LIN {X 0,Y 193.607,Z 643.258,A -85,B 0,C 180,E1 -26158.912,E2 -26158.912} C_VEL
LIN {X 0,Y 201.714,Z 651.879,A -85,B 0,C 180,E1 -26162.725,E2 -26162.725} C_VEL
LIN {X 0,Y 211.086,Z 659.54,A -85,B 0,C 180,E1 -26166.451,E2 -26166.451} C_VEL
LIN {X 0,Y 220.948,Z 665.783,A -85,B 0,C 180,E1 -26169.763,E2 -26169.763} C_VEL
LIN {X 0,Y 234.366,Z 672.498,A -85,B 0,C 180,E1 -26173.645,E2 -26173.645} C_VEL
LIN {X 0,Y 246.298,Z 677.555,A -85,B 0,C 180,E1 -26176.805,E2 -26176.805} C_VEL
LIN {X 0,Y 253.834,Z 680.558,A -85,B 0,C 180,E1 -26178.825,E2 -26178.825} C_VEL
LIN {X 0,Y 260.206,Z 683.111,A -85,B 0,C 180,E1 -26180.674,E2 -26180.674} C_VEL
LIN {X 0,Y 265.463,Z 685.211,A -85,B 0,C 180,E1 -26182.393,E2 -26182.393} C_VEL
LIN {X 0,Y 269.417,Z 686.886,A -85,B 0,C 180,E1 -26184.011,E2 -26184.011} C_VEL
LIN {X 0,Y 272.304,Z 688.198,A -85,B 0,C 180,E1 -26185.559,E2 -26185.559} C_VEL
LIN {X 0,Y 274.956,Z 689.105,A -85,B 0,C 180,E1 -26187.07,E2 -26187.07} C_VEL
LIN {X 0,Y 276.564,Z 689.664,A -85,B 0,C 180,E1 -26188.544,E2 -26188.544} C_VEL
LIN {X 0,Y 277.483,Z 689.842,A -85,B 0,C 180,E1 -26190,E2 -26190} C_VEL
LIN {X 0,Y 276.566,Z 689.663,A -85,B 0,C 180,E1 -26191.456,E2 -26191.456} C_VEL
LIN {X 0,Y 274.501,Z 688.974,A -85,B 0,C 180,E1 -26193.184,E2 -26193.184} C_VEL
LIN {X 0,Y 272.278,Z 688.199,A -85,B 0,C 180,E1 -26194.441,E2 -26194.441} C_VEL
LIN {X 0,Y 268.678,Z 686.595,A -85,B 0,C 180,E1 -26196.311,E2 -26196.311} C_VEL
LIN {X 0,Y 265.415,Z 685.213,A -85,B 0,C 180,E1 -26197.608,E2 -26197.608} C_VEL
LIN {X 0,Y 260.173,Z 683.112,A -85,B 0,C 180,E1 -26199.327,E2 -26199.327} C_VEL
LIN {X 0,Y 253.886,Z 680.557,A -85,B 0,C 180,E1 -26201.173,E2 -26201.173} C_VEL
LIN {X 0,Y 245.609,Z 677.259,A -85,B 0,C 180,E1 -26203.385,E2 -26203.385} C_VEL
LIN {X 0,Y 234.359,Z 672.513,A -85,B 0,C 180,E1 -26206.349,E2 -26206.349} C_VEL
LIN {X 0,Y 220.948,Z 665.784,A -85,B 0,C 180,E1 -26210.237,E2 -26210.237} C_VEL
LIN {X 0,Y 211.166,Z 659.537,A -85,B 0,C 180,E1 -26213.539,E2 -26213.539} C_VEL
LIN {X 0,Y 201.751,Z 651.903,A -85,B 0,C 180,E1 -26217.262,E2 -26217.262} C_VEL
LIN {X 0,Y 192.245,Z 641.559,A -85,B 0,C 180,E1 -26221.794,E2 -26221.794} C_VEL
LIN {X 0,Y 185.61,Z 632.244,A -85,B 0,C 180,E1 -26225.461,E2 -26225.461} C_VEL
LIN {X 0,Y 180.259,Z 622.941,A -85,B 0,C 180,E1 -26228.767,E2 -26228.767} C_VEL
LIN {X 0,Y 175.258,Z 612.247,A -85,B 0,C 180,E1 -26232.116,E2 -26232.116} C_VEL
LIN {X 0,Y 170.985,Z 601.587,A -85,B 0,C 180,E1 -26235.058,E2 -26235.058} C_VEL
LIN {X 0,Y 167.177,Z 590.937,A -85,B 0,C 180,E1 -26237.634,E2 -26237.634} C_VEL
LIN {X 0,Y 160.92,Z 572.907,A -85,B 0,C 180,E1 -26241.531,E2 -26241.531} C_VEL
LIN {X 0,Y 157.524,Z 564.607,A -85,B 0,C 180,E1 -26243.75,E2 -26243.75} C_VEL
LIN {X 0,Y 153.292,Z 555.729,A -85,B 0,C 180,E1 -26246.722,E2 -26246.722} C_VEL
LIN {X 0,Y 148.61,Z 547.106,A -85,B 0,C 180,E1 -26250.427,E2 -26250.427} C_VEL
LIN {X 0,Y 144.239,Z 539.962,A -85,B 0,C 180,E1 -26254.48,E2 -26254.48} C_VEL
LIN {X 0,Y 141.462,Z 535.851,A -85,B 0,C 180,E1 -26257.504,E2 -26257.504} C_VEL
LIN {X 0,Y 138.867,Z 531.989,A -85,B 0,C 180,E1 -26260.874,E2 -26260.874} C_VEL
LIN {X 0,Y 136.38,Z 528.521,A -85,B 0,C 180,E1 -26264.882,E2 -26264.882} C_VEL
LIN {X 0,Y 135.759,Z 527.362,A -85,B 0,C 180,E1 -26266.152,E2 -26266.152} C_VEL
LIN {X 0,Y 133.331,Z 524.419,A -85,B 0,C 180,E1 -26272.623,E2 -26272.623} C_VEL
LIN {X 0,Y 132.769,Z 522.602,A -85,B 0,C 180,E1 -26276.211,E2 -26276.211} C_VEL
LIN {X 0,Y 132.584,Z 521.985,A -85,B 0,C 180,E1 -26280.005,E2 -26280.005} C_VEL
LIN {X 0,Y 132.854,Z 522.928,A -85,B 0,C 180,E1 -26284.176,E2 -26284.176} C_VEL
LIN {X 0,Y 135.306,Z 527.03,A -85,B 0,C 180,E1 -26292.567,E2 -26292.567} C_VEL
LIN {X 0,Y 136.125,Z 527.942,A -85,B 0,C 180,E1 -26294.2,E2 -26294.2} C_VEL
LIN {X 0,Y 138.548,Z 531.658,A -85,B 0,C 180,E1 -26298.297,E2 -26298.297} C_VEL
LIN {X 0,Y 139.546,Z 533.014,A -85,B 0,C 180,E1 -26299.687,E2 -26299.687} C_VEL
LIN {X 0,Y 142.466,Z 537.271,A -85,B 0,C 180,E1 -26303.248,E2 -26303.248} C_VEL
LIN {X 0,Y 145.553,Z 542.106,A -85,B 0,C 180,E1 -26306.436,E2 -26306.436} C_VEL
LIN {X 0,Y 147.873,Z 546.115,A -85,B 0,C 180,E1 -26308.575,E2 -26308.575} C_VEL
LIN {X 0,Y 151.392,Z 554.209,A -85,B 0,C 180,E1 -26311.634,E2 -26311.634} C_VEL
LIN {X 0,Y 155.275,Z 564.625,A -85,B 0,C 180,E1 -26314.706,E2 -26314.706} C_VEL
LIN {X 0,Y 156.576,Z 568.776,A -85,B 0,C 180,E1 -26315.702,E2 -26315.702} C_VEL
LIN {X 0,Y 154.246,Z 595.965,A -85,B 0,C 180,E1 -26316.746,E2 -26316.746} C_VEL
LIN {X 0,Y 152.545,Z 606.818,A -85,B 0,C 180,E1 -26317.392,E2 -26317.392} C_VEL
LIN {X 0,Y 150.313,Z 616.609,A -85,B 0,C 180,E1 -26318.18,E2 -26318.18} C_VEL
LIN {X 0,Y 147.465,Z 626.405,A -85,B 0,C 180,E1 -26319.245,E2 -26319.245} C_VEL
LIN {X 0,Y 144.346,Z 635.167,A -85,B 0,C 180,E1 -26320.47,E2 -26320.47} C_VEL
LIN {X 0,Y 140.701,Z 643.886,A -85,B 0,C 180,E1 -26322.013,E2 -26322.013} C_VEL
LIN {X 0,Y 136.637,Z 652.394,A -85,B 0,C 180,E1 -26323.938,E2 -26323.938} C_VEL
LIN {X 0,Y 132.209,Z 660.562,A -85,B 0,C 180,E1 -26326.287,E2 -26326.287} C_VEL
LIN {X 0,Y 128.06,Z 667.504,A -85,B 0,C 180,E1 -26328.81,E2 -26328.81} C_VEL
LIN {X 0,Y 124.167,Z 673.491,A -85,B 0,C 180,E1 -26331.493,E2 -26331.493} C_VEL
LIN {X 0,Y 119.546,Z 680.2,A -85,B 0,C 180,E1 -26335.399,E2 -26335.399} C_VEL
LIN {X 0,Y 116.001,Z 685.08,A -85,B 0,C 180,E1 -26339.004,E2 -26339.004} C_VEL
LIN {X 0,Y 111.98,Z 690.174,A -85,B 0,C 180,E1 -26343.939,E2 -26343.939} C_VEL
LIN {X 0,Y 108.812,Z 694.141,A -85,B 0,C 180,E1 -26349.192,E2 -26349.192} C_VEL
LIN {X 0,Y 106.71,Z 697.085,A -85,B 0,C 180,E1 -26354.726,E2 -26354.726} C_VEL
LIN {X 0,Y 105.784,Z 698.592,A -85,B 0,C 180,E1 -26358.503,E2 -26358.503} C_VEL
LIN {X 0,Y 105.043,Z 700.131,A -85,B 0,C 180,E1 -26366.164,E2 -26366.164} C_VEL
LIN {X 0,Y 105.176,Z 700.418,A -85,B 0,C 180,E1 -26370,E2 -26370} C_VEL
LIN {X 0,Y 105.231,Z 699.528,A -85,B 0,C 180,E1 -26377.676,E2 -26377.676} C_VEL
LIN {X 0,Y 105.787,Z 698.592,A -85,B 0,C 180,E1 -26381.496,E2 -26381.496} C_VEL
LIN {X 0,Y 107.993,Z 695.232,A -85,B 0,C 180,E1 -26388.989,E2 -26388.989} C_VEL
LIN {X 0,Y 110.82,Z 691.602,A -85,B 0,C 180,E1 -26394.344,E2 -26394.344} C_VEL
LIN {X 0,Y 114.515,Z 686.868,A -85,B 0,C 180,E1 -26399.404,E2 -26399.404} C_VEL
LIN {X 0,Y 118.575,Z 681.494,A -85,B 0,C 180,E1 -26403.708,E2 -26403.708} C_VEL
LIN {X 0,Y 122.392,Z 676.116,A -85,B 0,C 180,E1 -26407.08,E2 -26407.08} C_VEL
LIN {X 0,Y 126.08,Z 670.624,A -85,B 0,C 180,E1 -26409.869,E2 -26409.869} C_VEL
LIN {X 0,Y 131.15,Z 662.411,A -85,B 0,C 180,E1 -26413.097,E2 -26413.097} C_VEL
LIN {X 0,Y 135.553,Z 654.591,A -85,B 0,C 180,E1 -26415.47,E2 -26415.47} C_VEL
LIN {X 0,Y 139.541,Z 646.511,A -85,B 0,C 180,E1 -26417.441,E2 -26417.441} C_VEL
LIN {X 0,Y 143.721,Z 636.756,A -85,B 0,C 180,E1 -26419.284,E2 -26419.284} C_VEL
LIN {X 0,Y 146.789,Z 628.37,A -85,B 0,C 180,E1 -26420.536,E2 -26420.536} C_VEL
LIN {X 0,Y 149.971,Z 617.87,A -85,B 0,C 180,E1 -26421.715,E2 -26421.715} C_VEL
LIN {X 0,Y 152.398,Z 607.507,A -85,B 0,C 180,E1 -26422.571,E2 -26422.571} C_VEL
LIN {X 0,Y 154.029,Z 597.554,A -85,B 0,C 180,E1 -26423.182,E2 -26423.182} C_VEL
LIN {X 0,Y 155.824,Z 578.344,A -85,B 0,C 180,E1 -26423.944,E2 -26423.944} C_VEL
LIN {X 0,Y 156.52,Z 568.606,A -85,B 0,C 180,E1 -26424.339,E2 -26424.339} C_VEL
LIN {X 0,Y 153.874,Z 560.714,A -85,B 0,C 180,E1 -26426.368,E2 -26426.368} C_VEL
LIN {X 0,Y 149.72,Z 550.16,A -85,B 0,C 180,E1 -26429.786,E2 -26429.786} C_VEL
LIN {X 0,Y 147.011,Z 544.436,A -85,B 0,C 180,E1 -26432.214,E2 -26432.214} C_VEL
LIN {X 0,Y 143.831,Z 539.389,A -85,B 0,C 180,E1 -26435.281,E2 -26435.281} C_VEL
LIN {X 0,Y 141.559,Z 535.941,A -85,B 0,C 180,E1 -26437.786,E2 -26437.786} C_VEL
LIN {X 0,Y 139.135,Z 532.246,A -85,B 0,C 180,E1 -26440.903,E2 -26440.903} C_VEL
LIN {X 0,Y 138.064,Z 531.159,A -85,B 0,C 180,E1 -26442.398,E2 -26442.398} C_VEL
LIN {X 0,Y 136.969,Z 530.727,A -85,B 0,C 180,E1 -26443.964,E2 -26443.964} C_VEL
LIN {X 0,Y 134.922,Z 531.049,A -85,B 0,C 180,E1 -26447.206,E2 -26447.206} C_VEL
LIN {X 0,Y 133.264,Z 531.693,A -85,B 0,C 180,E1 -26450.577,E2 -26450.577} C_VEL
LIN {X 0,Y 132.425,Z 531.436,A -85,B 0,C 180,E1 -26453.142,E2 -26453.142} C_VEL
LIN {X 0,Y 132.241,Z 531.075,A -85,B 0,C 180,E1 -26453.991,E2 -26453.991} C_VEL
LIN {X 0,Y 131.799,Z 529.387,A -85,B 0,C 180,E1 -26457.703,E2 -26457.703} C_VEL
LIN {X 0,Y 131.717,Z 529.047,A -85,B 0,C 180,E1 -26459.995,E2 -26459.995} C_VEL
LIN {X 0,Y 131.926,Z 529.956,A -85,B 0,C 180,E1 -26464.196,E2 -26464.196} C_VEL
LIN {X 0,Y 134.158,Z 533.971,A -85,B 0,C 180,E1 -26472.428,E2 -26472.428} C_VEL
LIN {X 0,Y 134.782,Z 534.696,A -85,B 0,C 180,E1 -26473.758,E2 -26473.758} C_VEL
LIN {X 0,Y 137.254,Z 538.568,A -85,B 0,C 180,E1 -26478.18,E2 -26478.18} C_VEL
LIN {X 0,Y 140.569,Z 543.731,A -85,B 0,C 180,E1 -26482.647,E2 -26482.647} C_VEL
LIN {X 0,Y 143.405,Z 548.348,A -85,B 0,C 180,E1 -26485.777,E2 -26485.777} C_VEL
LIN {X 0,Y 147.758,Z 556.106,A -85,B 0,C 180,E1 -26489.858,E2 -26489.858} C_VEL
LIN {X 0,Y 152.402,Z 565.552,A -85,B 0,C 180,E1 -26493.594,E2 -26493.594} C_VEL
LIN {X 0,Y 156.256,Z 574.926,A -85,B 0,C 180,E1 -26496.401,E2 -26496.401} C_VEL
LIN {X 0,Y 160.04,Z 586.179,A -85,B 0,C 180,E1 -26499.036,E2 -26499.036} C_VEL
LIN {X 0,Y 163.433,Z 597.185,A -85,B 0,C 180,E1 -26501.588,E2 -26501.588} C_VEL
LIN {X 0,Y 166.658,Z 607.047,A -85,B 0,C 180,E1 -26504.202,E2 -26504.202} C_VEL
LIN {X 0,Y 170.411,Z 617.155,A -85,B 0,C 180,E1 -26507.266,E2 -26507.266} C_VEL
LIN {X 0,Y 174.824,Z 627.17,A -85,B 0,C 180,E1 -26510.695,E2 -26510.695} C_VEL
LIN {X 0,Y 179.681,Z 635.973,A -85,B 0,C 180,E1 -26514.077,E2 -26514.077} C_VEL
LIN {X 0,Y 184.854,Z 643.572,A -85,B 0,C 180,E1 -26517.273,E2 -26517.273} C_VEL
LIN {X 0,Y 192.277,Z 652.277,A -85,B 0,C 180,E1 -26521.302,E2 -26521.302} C_VEL
LIN {X 0,Y 200.736,Z 659.845,A -85,B 0,C 180,E1 -26525.157,E2 -26525.157} C_VEL
LIN {X 0,Y 210.803,Z 666.663,A -85,B 0,C 180,E1 -26528.976,E2 -26528.976} C_VEL
LIN {X 0,Y 221.28,Z 672.126,A -85,B 0,C 180,E1 -26532.318,E2 -26532.318} C_VEL
LIN {X 0,Y 235.082,Z 677.867,A -85,B 0,C 180,E1 -26536.163,E2 -26536.163} C_VEL
LIN {X 0,Y 246.752,Z 682.108,A -85,B 0,C 180,E1 -26539.288,E2 -26539.288} C_VEL
LIN {X 0,Y 255.57,Z 685.165,A -85,B 0,C 180,E1 -26541.858,E2 -26541.858} C_VEL
LIN {X 0,Y 261.463,Z 687.257,A -85,B 0,C 180,E1 -26543.981,E2 -26543.981} C_VEL
LIN {X 0,Y 264.432,Z 688.418,A -85,B 0,C 180,E1 -26545.427,E2 -26545.427} C_VEL
LIN {X 0,Y 267.399,Z 689.359,A -85,B 0,C 180,E1 -26547.069,E2 -26547.069} C_VEL
LIN {X 0,Y 269.242,Z 689.867,A -85,B 0,C 180,E1 -26548.504,E2 -26548.504} C_VEL
LIN {X 0,Y 270.315,Z 690.041,A -85,B 0,C 180,E1 -26550,E2 -26550} C_VEL
LIN {X 0,Y 269.24,Z 689.867,A -85,B 0,C 180,E1 -26551.496,E2 -26551.496} C_VEL
LIN {X 0,Y 267.239,Z 689.317,A -85,B 0,C 180,E1 -26553.015,E2 -26553.015} C_VEL
LIN {X 0,Y 264.41,Z 688.418,A -85,B 0,C 180,E1 -26554.574,E2 -26554.574} C_VEL
LIN {X 0,Y 261.016,Z 687.117,A -85,B 0,C 180,E1 -26556.183,E2 -26556.183} C_VEL
LIN {X 0,Y 255.564,Z 685.178,A -85,B 0,C 180,E1 -26558.132,E2 -26558.132} C_VEL
LIN {X 0,Y 249.679,Z 683.135,A -85,B 0,C 180,E1 -26559.893,E2 -26559.893} C_VEL
LIN {X 0,Y 243.252,Z 680.857,A -85,B 0,C 180,E1 -26561.668,E2 -26561.668} C_VEL
LIN {X 0,Y 232.346,Z 676.846,A -85,B 0,C 180,E1 -26564.562,E2 -26564.562} C_VEL
LIN {X 0,Y 217.434,Z 670.286,A -85,B 0,C 180,E1 -26568.858,E2 -26568.858} C_VEL
LIN {X 0,Y 205.884,Z 663.53,A -85,B 0,C 180,E1 -26572.839,E2 -26572.839} C_VEL
LIN {X 0,Y 195.479,Z 655.394,A -85,B 0,C 180,E1 -26577.158,E2 -26577.158} C_VEL
LIN {X 0,Y 188.212,Z 647.778,A -85,B 0,C 180,E1 -26580.821,E2 -26580.821} C_VEL
LIN {X 0,Y 181.58,Z 639.028,A -85,B 0,C 180,E1 -26584.674,E2 -26584.674} C_VEL
LIN {X 0,Y 176.615,Z 630.661,A -85,B 0,C 180,E1 -26588.007,E2 -26588.007} C_VEL
LIN {X 0,Y 172.513,Z 622.049,A -85,B 0,C 180,E1 -26591.095,E2 -26591.095} C_VEL
LIN {X 0,Y 168.754,Z 612.855,A -85,B 0,C 180,E1 -26594.083,E2 -26594.083} C_VEL
LIN {X 0,Y 164.892,Z 601.852,A -85,B 0,C 180,E1 -26597.218,E2 -26597.218} C_VEL
LIN {X 0,Y 161.241,Z 590.184,A -85,B 0,C 180,E1 -26600.098,E2 -26600.098} C_VEL
LIN {X 0,Y 156.857,Z 576.56,A -85,B 0,C 180,E1 -26603.178,E2 -26603.178} C_VEL
LIN {X 0,Y 152.863,Z 566.622,A -85,B 0,C 180,E1 -26606.056,E2 -26606.056} C_VEL
LIN {X 0,Y 148.504,Z 557.612,A -85,B 0,C 180,E1 -26609.499,E2 -26609.499} C_VEL
LIN {X 0,Y 144.243,Z 549.708,A -85,B 0,C 180,E1 -26613.387,E2 -26613.387} C_VEL
LIN {X 0,Y 141.473,Z 545.217,A -85,B 0,C 180,E1 -26616.297,E2 -26616.297} C_VEL
LIN {X 0,Y 139.46,Z 542.029,A -85,B 0,C 180,E1 -26618.719,E2 -26618.719} C_VEL
LIN {X 0,Y 137.255,Z 538.56,A -85,B 0,C 180,E1 -26621.819,E2 -26621.819} C_VEL
LIN {X 0,Y 134.781,Z 534.7,A -85,B 0,C 180,E1 -26626.242,E2 -26626.242} C_VEL
LIN {X 0,Y 134.159,Z 533.961,A -85,B 0,C 180,E1 -26627.572,E2 -26627.572} C_VEL
LIN {X 0,Y 131.822,Z 529.519,A -85,B 0,C 180,E1 -26636.949,E2 -26636.949} C_VEL
LIN {X 0,Y 131.718,Z 529.04,A -85,B 0,C 180,E1 -26640.005,E2 -26640.005} C_VEL
LIN {X 0,Y 131.94,Z 529.991,A -85,B 0,C 180,E1 -26643.918,E2 -26643.918} C_VEL
LIN {X 0,Y 134.319,Z 534.061,A -85,B 0,C 180,E1 -26652.373,E2 -26652.373} C_VEL
LIN {X 0,Y 134.87,Z 534.887,A -85,B 0,C 180,E1 -26653.566,E2 -26653.566} C_VEL
LIN {X 0,Y 137.881,Z 539.509,A -85,B 0,C 180,E1 -26658.726,E2 -26658.726} C_VEL
LIN {X 0,Y 140.659,Z 543.824,A -85,B 0,C 180,E1 -26662.359,E2 -26662.359} C_VEL
LIN {X 0,Y 144.231,Z 549.666,A -85,B 0,C 180,E1 -26666.21,E2 -26666.21} C_VEL
LIN {X 0,Y 146.772,Z 555.356,A -85,B 0,C 180,E1 -26668.712,E2 -26668.712} C_VEL
LIN {X 0,Y 150.791,Z 566.153,A -85,B 0,C 180,E1 -26672.316,E2 -26672.316} C_VEL
LIN {X 0,Y 152.326,Z 571.077,A -85,B 0,C 180,E1 -26673.622,E2 -26673.622} C_VEL
LIN {X 0,Y 150.054,Z 596.194,A -85,B 0,C 180,E1 -26674.595,E2 -26674.595} C_VEL
LIN {X 0,Y 148.212,Z 607.312,A -85,B 0,C 180,E1 -26675.26,E2 -26675.26} C_VEL
LIN {X 0,Y 145.05,Z 620.182,A -85,B 0,C 180,E1 -26676.341,E2 -26676.341} C_VEL
LIN {X 0,Y 141.148,Z 631.794,A -85,B 0,C 180,E1 -26677.774,E2 -26677.774} C_VEL
LIN {X 0,Y 136.685,Z 642.378,A -85,B 0,C 180,E1 -26679.533,E2 -26679.533} C_VEL
LIN {X 0,Y 132.432,Z 651.101,A -85,B 0,C 180,E1 -26681.445,E2 -26681.445} C_VEL
LIN {X 0,Y 128.306,Z 658.516,A -85,B 0,C 180,E1 -26683.467,E2 -26683.467} C_VEL
LIN {X 0,Y 122.8,Z 667.308,A -85,B 0,C 180,E1 -26686.625,E2 -26686.625} C_VEL
LIN {X 0,Y 118.669,Z 673.294,A -85,B 0,C 180,E1 -26689.349,E2 -26689.349} C_VEL
LIN {X 0,Y 114.137,Z 679.517,A -85,B 0,C 180,E1 -26693.014,E2 -26693.014} C_VEL
LIN {X 0,Y 109.963,Z 684.884,A -85,B 0,C 180,E1 -26697.095,E2 -26697.095} C_VEL
LIN {X 0,Y 105.619,Z 689.977,A -85,B 0,C 180,E1 -26702.239,E2 -26702.239} C_VEL
LIN {X 0,Y 102.189,Z 693.944,A -85,B 0,C 180,E1 -26707.774,E2 -26707.774} C_VEL
LIN {X 0,Y 99.835,Z 696.887,A -85,B 0,C 180,E1 -26713.645,E2 -26713.645} C_VEL
LIN {X 0,Y 98.804,Z 698.395,A -85,B 0,C 180,E1 -26717.679,E2 -26717.679} C_VEL
LIN {X 0,Y 97.949,Z 699.935,A -85,B 0,C 180,E1 -26725.885,E2 -26725.885} C_VEL
LIN {X 0,Y 98.083,Z 700.222,A -85,B 0,C 180,E1 -26730,E2 -26730} C_VEL
LIN {X 0,Y 98.188,Z 699.331,A -85,B 0,C 180,E1 -26738.23,E2 -26738.23} C_VEL
LIN {X 0,Y 98.806,Z 698.395,A -85,B 0,C 180,E1 -26742.321,E2 -26742.321} C_VEL
LIN {X 0,Y 101.264,Z 695.034,A -85,B 0,C 180,E1 -26750.305,E2 -26750.305} C_VEL
LIN {X 0,Y 104.361,Z 691.405,A -85,B 0,C 180,E1 -26755.959,E2 -26755.959} C_VEL
LIN {X 0,Y 108.374,Z 686.672,A -85,B 0,C 180,E1 -26761.251,E2 -26761.251} C_VEL
LIN {X 0,Y 113.448,Z 680.404,A -85,B 0,C 180,E1 -26766.349,E2 -26766.349} C_VEL
LIN {X 0,Y 118.685,Z 673.295,A -85,B 0,C 180,E1 -26770.645,E2 -26770.645} C_VEL
LIN {X 0,Y 124.945,Z 664.064,A -85,B 0,C 180,E1 -26774.676,E2 -26774.676} C_VEL
LIN {X 0,Y 130.657,Z 654.394,A -85,B 0,C 180,E1 -26777.697,E2 -26777.697} C_VEL
LIN {X 0,Y 134.838,Z 646.315,A -85,B 0,C 180,E1 -26779.665,E2 -26779.665} C_VEL
LIN {X 0,Y 139.196,Z 636.56,A -85,B 0,C 180,E1 -26781.498,E2 -26781.498} C_VEL
LIN {X 0,Y 142.374,Z 628.173,A -85,B 0,C 180,E1 -26782.747,E2 -26782.747} C_VEL
LIN {X 0,Y 145.686,Z 617.674,A -85,B 0,C 180,E1 -26783.903,E2 -26783.903} C_VEL
LIN {X 0,Y 148.191,Z 607.313,A -85,B 0,C 180,E1 -26784.751,E2 -26784.751} C_VEL
LIN {X 0,Y 149.949,Z 596.931,A -85,B 0,C 180,E1 -26785.365,E2 -26785.365} C_VEL
LIN {X 0,Y 151.985,Z 575.616,A -85,B 0,C 180,E1 -26786.192,E2 -26786.192} C_VEL
LIN {X 0,Y 152.233,Z 570.793,A -85,B 0,C 180,E1 -26786.453,E2 -26786.453} C_VEL
LIN {X 0,Y 150.06,Z 564.182,A -85,B 0,C 180,E1 -26788.299,E2 -26788.299} C_VEL
LIN {X 0,Y 146.442,Z 554.498,A -85,B 0,C 180,E1 -26791.609,E2 -26791.609} C_VEL
LIN {X 0,Y 144.15,Z 549.512,A -85,B 0,C 180,E1 -26793.872,E2 -26793.872} C_VEL
LIN {X 0,Y 140.041,Z 542.737,A -85,B 0,C 180,E1 -26798.404,E2 -26798.404} C_VEL
LIN {X 0,Y 137.085,Z 538.343,A -85,B 0,C 180,E1 -26802.466,E2 -26802.466} C_VEL
LIN {X 0,Y 134.697,Z 534.461,A -85,B 0,C 180,E1 -26806.834,E2 -26806.834} C_VEL
LIN {X 0,Y 132.241,Z 531.075,A -85,B 0,C 180,E1 -26813.991,E2 -26813.991} C_VEL
LIN {X 0,Y 131.928,Z 530.66,A -85,B 0,C 180,E1 -26815.676,E2 -26815.676} C_VEL
LIN {X 0,Y 131.504,Z 531.404,A -85,B 0,C 180,E1 -26818.225,E2 -26818.225} C_VEL
LIN {X 0,Y 131.115,Z 534.724,A -85,B 0,C 180,E1 -26822.391,E2 -26822.391} C_VEL
LIN {X 0,Y 131.269,Z 537.711,A -85,B 0,C 180,E1 -26825.753,E2 -26825.753} C_VEL
LIN {X 0,Y 131.577,Z 538.823,A -85,B 0,C 180,E1 -26827.477,E2 -26827.477} C_VEL
LIN {X 0,Y 133.476,Z 541.439,A -85,B 0,C 180,E1 -26832.926,E2 -26832.926} C_VEL
LIN {X 0,Y 135.862,Z 545.334,A -85,B 0,C 180,E1 -26837.493,E2 -26837.493} C_VEL
LIN {X 0,Y 138.864,Z 550.396,A -85,B 0,C 180,E1 -26841.815,E2 -26841.815} C_VEL
LIN {X 0,Y 141.09,Z 554.185,A -85,B 0,C 180,E1 -26844.455,E2 -26844.455} C_VEL
LIN {X 0,Y 145.036,Z 561.671,A -85,B 0,C 180,E1 -26848.487,E2 -26848.487} C_VEL
LIN {X 0,Y 149.247,Z 570.719,A -85,B 0,C 180,E1 -26852.172,E2 -26852.172} C_VEL
LIN {X 0,Y 152.826,Z 579.943,A -85,B 0,C 180,E1 -26855.011,E2 -26855.011} C_VEL
LIN {X 0,Y 155.977,Z 590.349,A -85,B 0,C 180,E1 -26857.561,E2 -26857.561} C_VEL
LIN {X 0,Y 158.362,Z 599.183,A -85,B 0,C 180,E1 -26859.737,E2 -26859.737} C_VEL
LIN {X 0,Y 161.065,Z 608.7,A -85,B 0,C 180,E1 -26862.383,E2 -26862.383} C_VEL
LIN {X 0,Y 163.883,Z 617.554,A -85,B 0,C 180,E1 -26865.153,E2 -26865.153} C_VEL
LIN {X 0,Y 167.126,Z 626.218,A -85,B 0,C 180,E1 -26868.185,E2 -26868.185} C_VEL
LIN {X 0,Y 170.873,Z 634.482,A -85,B 0,C 180,E1 -26871.389,E2 -26871.389} C_VEL
LIN {X 0,Y 176.446,Z 644.006,A -85,B 0,C 180,E1 -26875.553,E2 -26875.553} C_VEL
LIN {X 0,Y 183.092,Z 652.655,A -85,B 0,C 180,E1 -26879.749,E2 -26879.749} C_VEL
LIN {X 0,Y 190.671,Z 660.146,A -85,B 0,C 180,E1 -26883.749,E2 -26883.749} C_VEL
LIN {X 0,Y 198.336,Z 665.908,A -85,B 0,C 180,E1 -26887.108,E2 -26887.108} C_VEL
LIN {X 0,Y 208.351,Z 671.711,A -85,B 0,C 180,E1 -26890.808,E2 -26890.808} C_VEL
LIN {X 0,Y 219.133,Z 676.52,A -85,B 0,C 180,E1 -26894.173,E2 -26894.173} C_VEL
LIN {X 0,Y 232.109,Z 681.172,A -85,B 0,C 180,E1 -26897.763,E2 -26897.763} C_VEL
LIN {X 0,Y 242.25,Z 684.363,A -85,B 0,C 180,E1 -26900.515,E2 -26900.515} C_VEL
LIN {X 0,Y 248.219,Z 686.173,A -85,B 0,C 180,E1 -26902.274,E2 -26902.274} C_VEL
LIN {X 0,Y 254.236,Z 687.958,A -85,B 0,C 180,E1 -26904.334,E2 -26904.334} C_VEL
LIN {X 0,Y 256.368,Z 688.643,A -85,B 0,C 180,E1 -26905.283,E2 -26905.283} C_VEL
LIN {X 0,Y 260.299,Z 689.748,A -85,B 0,C 180,E1 -26907.356,E2 -26907.356} C_VEL
LIN {X 0,Y 261.821,Z 690.072,A -85,B 0,C 180,E1 -26908.462,E2 -26908.462} C_VEL
LIN {X 0,Y 263.123,Z 690.239,A -85,B 0,C 180,E1 -26910,E2 -26910} C_VEL
LIN {X 0,Y 261.817,Z 690.071,A -85,B 0,C 180,E1 -26911.538,E2 -26911.538} C_VEL
LIN {X 0,Y 259.449,Z 689.531,A -85,B 0,C 180,E1 -26913.106,E2 -26913.106} C_VEL
LIN {X 0,Y 256.345,Z 688.643,A -85,B 0,C 180,E1 -26914.718,E2 -26914.718} C_VEL
LIN {X 0,Y 254.232,Z 687.965,A -85,B 0,C 180,E1 -26915.658,E2 -26915.658} C_VEL
LIN {X 0,Y 248.218,Z 686.176,A -85,B 0,C 180,E1 -26917.724,E2 -26917.724} C_VEL
LIN {X 0,Y 239.977,Z 683.679,A -85,B 0,C 180,E1 -26920.12,E2 -26920.12} C_VEL
LIN {X 0,Y 230.5,Z 680.631,A -85,B 0,C 180,E1 -26922.676,E2 -26922.676} C_VEL
LIN {X 0,Y 214.81,Z 674.704,A -85,B 0,C 180,E1 -26927.125,E2 -26927.125} C_VEL
LIN {X 0,Y 203.242,Z 668.921,A -85,B 0,C 180,E1 -26931,E2 -26931} C_VEL
LIN {X 0,Y 193.666,Z 662.535,A -85,B 0,C 180,E1 -26934.884,E2 -26934.884} C_VEL
LIN {X 0,Y 186.106,Z 655.804,A -85,B 0,C 180,E1 -26938.606,E2 -26938.606} C_VEL
LIN {X 0,Y 179.276,Z 647.971,A -85,B 0,C 180,E1 -26942.568,E2 -26942.568} C_VEL
LIN {X 0,Y 174.048,Z 640.217,A -85,B 0,C 180,E1 -26946.146,E2 -26946.146} C_VEL
LIN {X 0,Y 169.699,Z 632.112,A -85,B 0,C 180,E1 -26949.557,E2 -26949.557} C_VEL
LIN {X 0,Y 165.816,Z 622.857,A -85,B 0,C 180,E1 -26953.025,E2 -26953.025} C_VEL
LIN {X 0,Y 162.519,Z 613.253,A -85,B 0,C 180,E1 -26956.225,E2 -26956.225} C_VEL
LIN {X 0,Y 159.259,Z 602.507,A -85,B 0,C 180,E1 -26959.396,E2 -26959.396} C_VEL
LIN {X 0,Y 156.191,Z 591.08,A -85,B 0,C 180,E1 -26962.296,E2 -26962.296} C_VEL
LIN {X 0,Y 152.909,Z 580.112,A -85,B 0,C 180,E1 -26964.93,E2 -26964.93} C_VEL
LIN {X 0,Y 149.16,Z 570.549,A -85,B 0,C 180,E1 -26967.896,E2 -26967.896} C_VEL
LIN {X 0,Y 145.19,Z 562.04,A -85,B 0,C 180,E1 -26971.363,E2 -26971.363} C_VEL
LIN {X 0,Y 141.548,Z 554.977,A -85,B 0,C 180,E1 -26975.042,E2 -26975.042} C_VEL
LIN {X 0,Y 138.144,Z 549.065,A -85,B 0,C 180,E1 -26979.143,E2 -26979.143} C_VEL
LIN {X 0,Y 135.497,Z 544.882,A -85,B 0,C 180,E1 -26983.09,E2 -26983.09} C_VEL
LIN {X 0,Y 133.157,Z 540.966,A -85,B 0,C 180,E1 -26987.817,E2 -26987.817} C_VEL
LIN {X 0,Y 131.111,Z 537.419,A -85,B 0,C 180,E1 -26995.2,E2 -26995.2} C_VEL
LIN {X 0,Y 130.897,Z 536.44,A -85,B 0,C 180,E1 -26997.697,E2 -26997.697} C_VEL
LIN {X 0,Y 130.857,Z 536.195,A -85,B 0,C 180,E1 -27000.774,E2 -27000.774} C_VEL
LIN {X 0,Y 131.03,Z 537.046,A -85,B 0,C 180,E1 -27003.657,E2 -27003.657} C_VEL
LIN {X 0,Y 133.164,Z 540.952,A -85,B 0,C 180,E1 -27011.805,E2 -27011.805} C_VEL
LIN {X 0,Y 136.198,Z 545.92,A -85,B 0,C 180,E1 -27017.652,E2 -27017.652} C_VEL
LIN {X 0,Y 138.95,Z 550.524,A -85,B 0,C 180,E1 -27021.532,E2 -27021.532} C_VEL
LIN {X 0,Y 141.931,Z 555.68,A -85,B 0,C 180,E1 -27024.984,E2 -27024.984} C_VEL
LIN {X 0,Y 144.41,Z 561.744,A -85,B 0,C 180,E1 -27027.641,E2 -27027.641} C_VEL
LIN {X 0,Y 148.057,Z 572.635,A -85,B 0,C 180,E1 -27031.213,E2 -27031.213} C_VEL
LIN {X 0,Y 148.279,Z 573.652,A -85,B 0,C 180,E1 -27031.445,E2 -27031.445} C_VEL
LIN {X 0,Y 146.054,Z 596.712,A -85,B 0,C 180,E1 -27032.341,E2 -27032.341} C_VEL
LIN {X 0,Y 143.762,Z 609.216,A -85,B 0,C 180,E1 -27033.062,E2 -27033.062} C_VEL
LIN {X 0,Y 140.277,Z 622.078,A -85,B 0,C 180,E1 -27034.243,E2 -27034.243} C_VEL
LIN {X 0,Y 136.241,Z 633.187,A -85,B 0,C 180,E1 -27035.664,E2 -27035.664} C_VEL
LIN {X 0,Y 132.27,Z 642.182,A -85,B 0,C 180,E1 -27037.156,E2 -27037.156} C_VEL
LIN {X 0,Y 127.84,Z 650.904,A -85,B 0,C 180,E1 -27039.057,E2 -27039.057} C_VEL
LIN {X 0,Y 123.528,Z 658.32,A -85,B 0,C 180,E1 -27041.076,E2 -27041.076} C_VEL
LIN {X 0,Y 117.73,Z 667.111,A -85,B 0,C 180,E1 -27044.247,E2 -27044.247} C_VEL
LIN {X 0,Y 113.364,Z 673.098,A -85,B 0,C 180,E1 -27047.005,E2 -27047.005} C_VEL
LIN {X 0,Y 108.255,Z 679.629,A -85,B 0,C 180,E1 -27050.971,E2 -27050.971} C_VEL
LIN {X 0,Y 104.056,Z 684.687,A -85,B 0,C 180,E1 -27054.964,E2 -27054.964} C_VEL
LIN {X 0,Y 99.35,Z 689.779,A -85,B 0,C 180,E1 -27060.319,E2 -27060.319} C_VEL
LIN {X 0,Y 95.616,Z 693.746,A -85,B 0,C 180,E1 -27066.155,E2 -27066.155} C_VEL
LIN {X 0,Y 93.01,Z 696.69,A -85,B 0,C 180,E1 -27072.408,E2 -27072.408} C_VEL
LIN {X 0,Y 91.857,Z 698.198,A -85,B 0,C 180,E1 -27076.731,E2 -27076.731} C_VEL
LIN {X 0,Y 90.879,Z 699.739,A -85,B 0,C 180,E1 -27085.565,E2 -27085.565} C_VEL
LIN {X 0,Y 90.981,Z 700.026,A -85,B 0,C 180,E1 -27090,E2 -27090} C_VEL
LIN {X 0,Y 91.149,Z 699.134,A -85,B 0,C 180,E1 -27098.871,E2 -27098.871} C_VEL
LIN {X 0,Y 91.859,Z 698.198,A -85,B 0,C 180,E1 -27103.269,E2 -27103.269} C_VEL
LIN {X 0,Y 94.601,Z 694.837,A -85,B 0,C 180,E1 -27111.805,E2 -27111.805} C_VEL
LIN {X 0,Y 98.001,Z 691.208,A -85,B 0,C 180,E1 -27117.784,E2 -27117.784} C_VEL
LIN {X 0,Y 102.362,Z 686.475,A -85,B 0,C 180,E1 -27123.316,E2 -27123.316} C_VEL
LIN {X 0,Y 105.72,Z 682.688,A -85,B 0,C 180,E1 -27126.748,E2 -27126.748} C_VEL
LIN {X 0,Y 110.348,Z 677.033,A -85,B 0,C 180,E1 -27130.754,E2 -27130.754} C_VEL
LIN {X 0,Y 115.511,Z 670.231,A -85,B 0,C 180,E1 -27134.402,E2 -27134.402} C_VEL
LIN {X 0,Y 121.15,Z 662.018,A -85,B 0,C 180,E1 -27137.7,E2 -27137.7} C_VEL
LIN {X 0,Y 125.969,Z 654.197,A -85,B 0,C 180,E1 -27140.096,E2 -27140.096} C_VEL
LIN {X 0,Y 130.359,Z 646.119,A -85,B 0,C 180,E1 -27142.042,E2 -27142.042} C_VEL
LIN {X 0,Y 134.897,Z 636.364,A -85,B 0,C 180,E1 -27143.855,E2 -27143.855} C_VEL
LIN {X 0,Y 138.201,Z 627.978,A -85,B 0,C 180,E1 -27145.085,E2 -27145.085} C_VEL
LIN {X 0,Y 141.624,Z 617.478,A -85,B 0,C 180,E1 -27146.222,E2 -27146.222} C_VEL
LIN {X 0,Y 144.289,Z 606.703,A -85,B 0,C 180,E1 -27147.084,E2 -27147.084} C_VEL
LIN {X 0,Y 146.053,Z 596.619,A -85,B 0,C 180,E1 -27147.658,E2 -27147.658} C_VEL
LIN {X 0,Y 148.301,Z 573.653,A -85,B 0,C 180,E1 -27148.541,E2 -27148.541} C_VEL
LIN {X 0,Y 146.446,Z 567.698,A -85,B 0,C 180,E1 -27150.308,E2 -27150.308} C_VEL
LIN {X 0,Y 143.238,Z 558.686,A -85,B 0,C 180,E1 -27153.594,E2 -27153.594} C_VEL
LIN {X 0,Y 141.591,Z 555.062,A -85,B 0,C 180,E1 -27155.383,E2 -27155.383} C_VEL
LIN {X 0,Y 138.221,Z 549.136,A -85,B 0,C 180,E1 -27159.438,E2 -27159.438} C_VEL
LIN {X 0,Y 135.425,Z 544.757,A -85,B 0,C 180,E1 -27163.604,E2 -27163.604} C_VEL
LIN {X 0,Y 133.164,Z 540.956,A -85,B 0,C 180,E1 -27168.195,E2 -27168.195} C_VEL
LIN {X 0,Y 130.929,Z 536.476,A -85,B 0,C 180,E1 -27177.688,E2 -27177.688} C_VEL
LIN {X 0,Y 130.85,Z 536.104,A -85,B 0,C 180,E1 -27179.995,E2 -27179.995} C_VEL
LIN {X 0,Y 131.01,Z 536.957,A -85,B 0,C 180,E1 -27183.84,E2 -27183.84} C_VEL
LIN {X 0,Y 131.577,Z 538.823,A -85,B 0,C 180,E1 -27187.477,E2 -27187.477} C_VEL
LIN {X 0,Y 132.155,Z 540.813,A -85,B 0,C 180,E1 -27189.879,E2 -27189.879} C_VEL
LIN {X 0,Y 132.755,Z 543.802,A -85,B 0,C 180,E1 -27192.089,E2 -27192.089} C_VEL
LIN {X 0,Y 134.999,Z 552.96,A -85,B 0,C 180,E1 -27197.653,E2 -27197.653} C_VEL
LIN {X 0,Y 135.902,Z 554.772,A -85,B 0,C 180,E1 -27199.118,E2 -27199.118} C_VEL
LIN {X 0,Y 138.848,Z 560.065,A -85,B 0,C 180,E1 -27203.091,E2 -27203.091} C_VEL
LIN {X 0,Y 142.353,Z 567.11,A -85,B 0,C 180,E1 -27207.012,E2 -27207.012} C_VEL
LIN {X 0,Y 146.12,Z 575.678,A -85,B 0,C 180,E1 -27210.626,E2 -27210.626} C_VEL
LIN {X 0,Y 149.459,Z 584.877,A -85,B 0,C 180,E1 -27213.535,E2 -27213.535} C_VEL
LIN {X 0,Y 152.698,Z 597.823,A -85,B 0,C 180,E1 -27216.848,E2 -27216.848} C_VEL
LIN {X 0,Y 154.993,Z 607.529,A -85,B 0,C 180,E1 -27219.571,E2 -27219.571} C_VEL
LIN {X 0,Y 157.42,Z 616.864,A -85,B 0,C 180,E1 -27222.533,E2 -27222.533} C_VEL
LIN {X 0,Y 160.547,Z 627.138,A -85,B 0,C 180,E1 -27226.236,E2 -27226.236} C_VEL
LIN {X 0,Y 164.211,Z 636.496,A -85,B 0,C 180,E1 -27230.061,E2 -27230.061} C_VEL
LIN {X 0,Y 168.342,Z 644.366,A -85,B 0,C 180,E1 -27233.671,E2 -27233.671} C_VEL
LIN {X 0,Y 174.097,Z 652.807,A -85,B 0,C 180,E1 -27237.958,E2 -27237.958} C_VEL
LIN {X 0,Y 181.057,Z 660.437,A -85,B 0,C 180,E1 -27242.239,E2 -27242.239} C_VEL
LIN {X 0,Y 189.316,Z 667.107,A -85,B 0,C 180,E1 -27246.372,E2 -27246.372} C_VEL
LIN {X 0,Y 198.155,Z 672.483,A -85,B 0,C 180,E1 -27250.02,E2 -27250.02} C_VEL
LIN {X 0,Y 208.731,Z 677.329,A -85,B 0,C 180,E1 -27253.645,E2 -27253.645} C_VEL
LIN {X 0,Y 222.918,Z 682.217,A -85,B 0,C 180,E1 -27257.765,E2 -27257.765} C_VEL
LIN {X 0,Y 228.928,Z 683.991,A -85,B 0,C 180,E1 -27259.386,E2 -27259.386} C_VEL
LIN {X 0,Y 236.566,Z 686.005,A -85,B 0,C 180,E1 -27261.458,E2 -27261.458} C_VEL
LIN {X 0,Y 242.966,Z 687.615,A -85,B 0,C 180,E1 -27263.356,E2 -27263.356} C_VEL
LIN {X 0,Y 248.091,Z 688.874,A -85,B 0,C 180,E1 -27265.125,E2 -27265.125} C_VEL
LIN {X 0,Y 253.206,Z 690.072,A -85,B 0,C 180,E1 -27267.655,E2 -27267.655} C_VEL
LIN {X 0,Y 254.33,Z 690.277,A -85,B 0,C 180,E1 -27268.417,E2 -27268.417} C_VEL
LIN {X 0,Y 255.899,Z 690.439,A -85,B 0,C 180,E1 -27270,E2 -27270} C_VEL
LIN {X 0,Y 254.324,Z 690.277,A -85,B 0,C 180,E1 -27271.583,E2 -27271.583} C_VEL
LIN {X 0,Y 251.531,Z 689.748,A -85,B 0,C 180,E1 -27273.203,E2 -27273.203} C_VEL
LIN {X 0,Y 248.07,Z 688.874,A -85,B 0,C 180,E1 -27274.876,E2 -27274.876} C_VEL
LIN {X 0,Y 240.884,Z 687.129,A -85,B 0,C 180,E1 -27277.288,E2 -27277.288} C_VEL
LIN {X 0,Y 234.82,Z 685.533,A -85,B 0,C 180,E1 -27279.03,E2 -27279.03} C_VEL
LIN {X 0,Y 228.825,Z 683.946,A -85,B 0,C 180,E1 -27280.652,E2 -27280.652} C_VEL
LIN {X 0,Y 217.138,Z 680.417,A -85,B 0,C 180,E1 -27283.848,E2 -27283.848} C_VEL
LIN {X 0,Y 203.352,Z 675.034,A -85,B 0,C 180,E1 -27288.122,E2 -27288.122} C_VEL
LIN {X 0,Y 193.756,Z 669.986,A -85,B 0,C 180,E1 -27291.734,E2 -27291.734} C_VEL
LIN {X 0,Y 184.021,Z 663.092,A -85,B 0,C 180,E1 -27296.178,E2 -27296.178} C_VEL
LIN {X 0,Y 176.901,Z 656.129,A -85,B 0,C 180,E1 -27300.23,E2 -27300.23} C_VEL
LIN {X 0,Y 170.576,Z 648.064,A -85,B 0,C 180,E1 -27304.517,E2 -27304.517} C_VEL
LIN {X 0,Y 165.878,Z 639.955,A -85,B 0,C 180,E1 -27308.396,E2 -27308.396} C_VEL
LIN {X 0,Y 162.12,Z 631.327,A -85,B 0,C 180,E1 -27312.088,E2 -27312.088} C_VEL
LIN {X 0,Y 158.928,Z 622.166,A -85,B 0,C 180,E1 -27315.612,E2 -27315.612} C_VEL
LIN {X 0,Y 156.235,Z 612.579,A -85,B 0,C 180,E1 -27318.869,E2 -27318.869} C_VEL
LIN {X 0,Y 153.76,Z 602.382,A -85,B 0,C 180,E1 -27321.904,E2 -27321.904} C_VEL
LIN {X 0,Y 151.316,Z 591.592,A -85,B 0,C 180,E1 -27324.719,E2 -27324.719} C_VEL
LIN {X 0,Y 148.543,Z 582.164,A -85,B 0,C 180,E1 -27327.244,E2 -27327.244} C_VEL
LIN {X 0,Y 145.153,Z 573.427,A -85,B 0,C 180,E1 -27330.251,E2 -27330.251} C_VEL
LIN {X 0,Y 141.601,Z 565.559,A -85,B 0,C 180,E1 -27333.771,E2 -27333.771} C_VEL
LIN {X 0,Y 138.095,Z 558.582,A -85,B 0,C 180,E1 -27337.861,E2 -27337.861} C_VEL
LIN {X 0,Y 135.718,Z 554.473,A -85,B 0,C 180,E1 -27341.159,E2 -27341.159} C_VEL
LIN {X 0,Y 134.115,Z 551.634,A -85,B 0,C 180,E1 -27343.841,E2 -27343.841} C_VEL
LIN {X 0,Y 131.983,Z 547.826,A -85,B 0,C 180,E1 -27348.475,E2 -27348.475} C_VEL
LIN {X 0,Y 130.115,Z 544.039,A -85,B 0,C 180,E1 -27356.327,E2 -27356.327} C_VEL
LIN {X 0,Y 129.979,Z 543.251,A -85,B 0,C 180,E1 -27359.23,E2 -27359.23} C_VEL
LIN {X 0,Y 130.054,Z 543.611,A -85,B 0,C 180,E1 -27362.328,E2 -27362.328} C_VEL
LIN {X 0,Y 132.278,Z 548.331,A -85,B 0,C 180,E1 -27371.886,E2 -27371.886} C_VEL
LIN {X 0,Y 134.823,Z 552.841,A -85,B 0,C 180,E1 -27377.005,E2 -27377.005} C_VEL
LIN {X 0,Y 137.228,Z 557.096,A -85,B 0,C 180,E1 -27380.62,E2 -27380.62} C_VEL
LIN {X 0,Y 139.931,Z 562.171,A -85,B 0,C 180,E1 -27383.99,E2 -27383.99} C_VEL
LIN {X 0,Y 142.331,Z 569.087,A -85,B 0,C 180,E1 -27386.822,E2 -27386.822} C_VEL
LIN {X 0,Y 144.462,Z 575.847,A -85,B 0,C 180,E1 -27389.115,E2 -27389.115} C_VEL
LIN {X 0,Y 142.341,Z 596.788,A -85,B 0,C 180,E1 -27389.935,E2 -27389.935} C_VEL
LIN {X 0,Y 139.742,Z 610.3,A -85,B 0,C 180,E1 -27390.723,E2 -27390.723} C_VEL
LIN {X 0,Y 136.403,Z 621.882,A -85,B 0,C 180,E1 -27391.774,E2 -27391.774} C_VEL
LIN {X 0,Y 132.229,Z 632.991,A -85,B 0,C 180,E1 -27393.165,E2 -27393.165} C_VEL
LIN {X 0,Y 128.105,Z 641.986,A -85,B 0,C 180,E1 -27394.623,E2 -27394.623} C_VEL
LIN {X 0,Y 123.481,Z 650.708,A -85,B 0,C 180,E1 -27396.493,E2 -27396.493} C_VEL
LIN {X 0,Y 118.982,Z 658.124,A -85,B 0,C 180,E1 -27398.497,E2 -27398.497} C_VEL
LIN {X 0,Y 112.861,Z 666.914,A -85,B 0,C 180,E1 -27401.648,E2 -27401.648} C_VEL
LIN {X 0,Y 108.259,Z 672.901,A -85,B 0,C 180,E1 -27404.431,E2 -27404.431} C_VEL
LIN {X 0,Y 102.573,Z 679.685,A -85,B 0,C 180,E1 -27408.652,E2 -27408.652} C_VEL
LIN {X 0,Y 98.291,Z 684.489,A -85,B 0,C 180,E1 -27412.572,E2 -27412.572} C_VEL
LIN {X 0,Y 93.209,Z 689.582,A -85,B 0,C 180,E1 -27418.143,E2 -27418.143} C_VEL
LIN {X 0,Y 89.14,Z 693.549,A -85,B 0,C 180,E1 -27424.302,E2 -27424.302} C_VEL
LIN {X 0,Y 86.243,Z 696.493,A -85,B 0,C 180,E1 -27430.976,E2 -27430.976} C_VEL
LIN {X 0,Y 84.949,Z 698.001,A -85,B 0,C 180,E1 -27435.629,E2 -27435.629} C_VEL
LIN {X 0,Y 83.795,Z 699.542,A -85,B 0,C 180,E1 -27445.189,E2 -27445.189} C_VEL
LIN {X 0,Y 83.888,Z 699.83,A -85,B 0,C 180,E1 -27450,E2 -27450} C_VEL
LIN {X 0,Y 84.136,Z 698.938,A -85,B 0,C 180,E1 -27459.617,E2 -27459.617} C_VEL
LIN {X 0,Y 84.95,Z 698.001,A -85,B 0,C 180,E1 -27464.37,E2 -27464.37} C_VEL
LIN {X 0,Y 88.012,Z 694.64,A -85,B 0,C 180,E1 -27473.532,E2 -27473.532} C_VEL
LIN {X 0,Y 91.754,Z 691.011,A -85,B 0,C 180,E1 -27479.859,E2 -27479.859} C_VEL
LIN {X 0,Y 96.5,Z 686.279,A -85,B 0,C 180,E1 -27485.635,E2 -27485.635} C_VEL
LIN {X 0,Y 100.095,Z 682.491,A -85,B 0,C 180,E1 -27489.191,E2 -27489.191} C_VEL
LIN {X 0,Y 105.043,Z 676.836,A -85,B 0,C 180,E1 -27493.297,E2 -27493.297} C_VEL
LIN {X 0,Y 110.528,Z 670.033,A -85,B 0,C 180,E1 -27496.989,E2 -27496.989} C_VEL
LIN {X 0,Y 116.474,Z 661.821,A -85,B 0,C 180,E1 -27500.293,E2 -27500.293} C_VEL
LIN {X 0,Y 121.523,Z 654,A -85,B 0,C 180,E1 -27502.673,E2 -27502.673} C_VEL
LIN {X 0,Y 126.105,Z 645.922,A -85,B 0,C 180,E1 -27504.593,E2 -27504.593} C_VEL
LIN {X 0,Y 130.84,Z 636.168,A -85,B 0,C 180,E1 -27506.363,E2 -27506.363} C_VEL
LIN {X 0,Y 134.274,Z 627.782,A -85,B 0,C 180,E1 -27507.564,E2 -27507.564} C_VEL
LIN {X 0,Y 137.809,Z 617.282,A -85,B 0,C 180,E1 -27508.672,E2 -27508.672} C_VEL
LIN {X 0,Y 140.471,Z 606.952,A -85,B 0,C 180,E1 -27509.482,E2 -27509.482} C_VEL
LIN {X 0,Y 142.47,Z 595.892,A -85,B 0,C 180,E1 -27510.083,E2 -27510.083} C_VEL
LIN {X 0,Y 144.462,Z 575.85,A -85,B 0,C 180,E1 -27510.885,E2 -27510.885} C_VEL
LIN {X 0,Y 141.046,Z 565.171,A -85,B 0,C 180,E1 -27514.67,E2 -27514.67} C_VEL
LIN {X 0,Y 139.403,Z 561.062,A -85,B 0,C 180,E1 -27516.637,E2 -27516.637} C_VEL
LIN {X 0,Y 136.361,Z 555.416,A -85,B 0,C 180,E1 -27520.618,E2 -27520.618} C_VEL
LIN {X 0,Y 133.917,Z 551.33,A -85,B 0,C 180,E1 -27524.588,E2 -27524.588} C_VEL
LIN {X 0,Y 131.984,Z 547.805,A -85,B 0,C 180,E1 -27528.866,E2 -27528.866} C_VEL
LIN {X 0,Y 130.017,Z 543.376,A -85,B 0,C 180,E1 -27538.447,E2 -27538.447} C_VEL
LIN {X 0,Y 129.984,Z 543.161,A -85,B 0,C 180,E1 -27539.995,E2 -27539.995} C_VEL
LIN {X 0,Y 130.1,Z 543.949,A -85,B 0,C 180,E1 -27543.479,E2 -27543.479} C_VEL
LIN {X 0,Y 131.983,Z 547.824,A -85,B 0,C 180,E1 -27551.525,E2 -27551.525} C_VEL
LIN {X 0,Y 134.764,Z 552.764,A -85,B 0,C 180,E1 -27557.298,E2 -27557.298} C_VEL
LIN {X 0,Y 135.902,Z 554.772,A -85,B 0,C 180,E1 -27559.118,E2 -27559.118} C_VEL
LIN {X 0,Y 136.818,Z 556.71,A -85,B 0,C 180,E1 -27560.495,E2 -27560.495} C_VEL
LIN {X 0,Y 137.95,Z 560.653,A -85,B 0,C 180,E1 -27562.272,E2 -27562.272} C_VEL
LIN {X 0,Y 140.934,Z 574.929,A -85,B 0,C 180,E1 -27566.735,E2 -27566.735} C_VEL
LIN {X 0,Y 141.942,Z 577.75,A -85,B 0,C 180,E1 -27567.841,E2 -27567.841} C_VEL
LIN {X 0,Y 145.012,Z 586.078,A -85,B 0,C 180,E1 -27570.887,E2 -27570.887} C_VEL
LIN {X 0,Y 147.331,Z 595.145,A -85,B 0,C 180,E1 -27573.468,E2 -27573.468} C_VEL
LIN {X 0,Y 149.66,Z 607.767,A -85,B 0,C 180,E1 -27577.031,E2 -27577.031} C_VEL
LIN {X 0,Y 151.755,Z 618.104,A -85,B 0,C 180,E1 -27580.412,E2 -27580.412} C_VEL
LIN {X 0,Y 154.171,Z 627.768,A -85,B 0,C 180,E1 -27584.036,E2 -27584.036} C_VEL
LIN {X 0,Y 157.069,Z 636.756,A -85,B 0,C 180,E1 -27587.843,E2 -27587.843} C_VEL
LIN {X 0,Y 160.774,Z 645.223,A -85,B 0,C 180,E1 -27591.884,E2 -27591.884} C_VEL
LIN {X 0,Y 165.69,Z 653.429,A -85,B 0,C 180,E1 -27596.262,E2 -27596.262} C_VEL
LIN {X 0,Y 171.724,Z 660.723,A -85,B 0,C 180,E1 -27600.587,E2 -27600.587} C_VEL
LIN {X 0,Y 178.753,Z 667.08,A -85,B 0,C 180,E1 -27604.718,E2 -27604.718} C_VEL
LIN {X 0,Y 188.048,Z 673.172,A -85,B 0,C 180,E1 -27609.11,E2 -27609.11} C_VEL
LIN {X 0,Y 198.366,Z 678.082,A -85,B 0,C 180,E1 -27613.043,E2 -27613.043} C_VEL
LIN {X 0,Y 209.527,Z 682.025,A -85,B 0,C 180,E1 -27616.571,E2 -27616.571} C_VEL
LIN {X 0,Y 221.303,Z 685.27,A -85,B 0,C 180,E1 -27619.872,E2 -27619.872} C_VEL
LIN {X 0,Y 227.378,Z 686.696,A -85,B 0,C 180,E1 -27621.502,E2 -27621.502} C_VEL
LIN {X 0,Y 233.541,Z 687.997,A -85,B 0,C 180,E1 -27623.225,E2 -27623.225} C_VEL
LIN {X 0,Y 239.783,Z 689.27,A -85,B 0,C 180,E1 -27625.188,E2 -27625.188} C_VEL
LIN {X 0,Y 243.466,Z 689.97,A -85,B 0,C 180,E1 -27626.69,E2 -27626.69} C_VEL
LIN {X 0,Y 246.785,Z 690.483,A -85,B 0,C 180,E1 -27628.368,E2 -27628.368} C_VEL
LIN {X 0,Y 248.629,Z 690.64,A -85,B 0,C 180,E1 -27630,E2 -27630} C_VEL
LIN {X 0,Y 246.77,Z 690.483,A -85,B 0,C 180,E1 -27631.632,E2 -27631.632} C_VEL
LIN {X 0,Y 243.446,Z 689.97,A -85,B 0,C 180,E1 -27633.31,E2 -27633.31} C_VEL
LIN {X 0,Y 239.017,Z 689.127,A -85,B 0,C 180,E1 -27635.061,E2 -27635.061} C_VEL
LIN {X 0,Y 233.045,Z 687.888,A -85,B 0,C 180,E1 -27636.928,E2 -27636.928} C_VEL
LIN {X 0,Y 225.677,Z 686.303,A -85,B 0,C 180,E1 -27638.958,E2 -27638.958} C_VEL
LIN {X 0,Y 215.345,Z 683.738,A -85,B 0,C 180,E1 -27641.758,E2 -27641.758} C_VEL
LIN {X 0,Y 200.328,Z 678.839,A -85,B 0,C 180,E1 -27646.299,E2 -27646.299} C_VEL
LIN {X 0,Y 190.875,Z 674.663,A -85,B 0,C 180,E1 -27649.74,E2 -27649.74} C_VEL
LIN {X 0,Y 180.97,Z 668.719,A -85,B 0,C 180,E1 -27654.139,E2 -27654.139} C_VEL
LIN {X 0,Y 174.565,Z 663.484,A -85,B 0,C 180,E1 -27657.669,E2 -27657.669} C_VEL
LIN {X 0,Y 167.914,Z 656.342,A -85,B 0,C 180,E1 -27662.061,E2 -27662.061} C_VEL
LIN {X 0,Y 162.977,Z 649.219,A -85,B 0,C 180,E1 -27666.054,E2 -27666.054} C_VEL
LIN {X 0,Y 158.836,Z 641.155,A -85,B 0,C 180,E1 -27670.131,E2 -27670.131} C_VEL
LIN {X 0,Y 155.328,Z 631.655,A -85,B 0,C 180,E1 -27674.372,E2 -27674.372} C_VEL
LIN {X 0,Y 153.056,Z 623.495,A -85,B 0,C 180,E1 -27677.629,E2 -27677.629} C_VEL
LIN {X 0,Y 150.603,Z 612.67,A -85,B 0,C 180,E1 -27681.419,E2 -27681.419} C_VEL
LIN {X 0,Y 148.586,Z 602.22,A -85,B 0,C 180,E1 -27684.595,E2 -27684.595} C_VEL
LIN {X 0,Y 146.49,Z 591.335,A -85,B 0,C 180,E1 -27687.544,E2 -27687.544} C_VEL
LIN {X 0,Y 144.002,Z 583.221,A -85,B 0,C 180,E1 -27690.09,E2 -27690.09} C_VEL
LIN {X 0,Y 141.196,Z 575.926,A -85,B 0,C 180,E1 -27692.943,E2 -27692.943} C_VEL
LIN {X 0,Y 138.104,Z 568.951,A -85,B 0,C 180,E1 -27696.479,E2 -27696.479} C_VEL
LIN {X 0,Y 135.58,Z 563.779,A -85,B 0,C 180,E1 -27699.865,E2 -27699.865} C_VEL
LIN {X 0,Y 133.692,Z 560.262,A -85,B 0,C 180,E1 -27702.855,E2 -27702.855} C_VEL
LIN {X 0,Y 132.445,Z 557.922,A -85,B 0,C 180,E1 -27705.21,E2 -27705.21} C_VEL
LIN {X 0,Y 130.827,Z 554.678,A -85,B 0,C 180,E1 -27709.144,E2 -27709.144} C_VEL
LIN {X 0,Y 129.126,Z 550.435,A -85,B 0,C 180,E1 -27718.445,E2 -27718.445} C_VEL
LIN {X 0,Y 129.122,Z 550.326,A -85,B 0,C 180,E1 -27720.784,E2 -27720.784} C_VEL
LIN {X 0,Y 129.306,Z 551.765,A -85,B 0,C 180,E1 -27724.193,E2 -27724.193} C_VEL
LIN {X 0,Y 131.092,Z 555.212,A -85,B 0,C 180,E1 -27731.211,E2 -27731.211} C_VEL
LIN {X 0,Y 133.318,Z 559.466,A -85,B 0,C 180,E1 -27736.072,E2 -27736.072} C_VEL
LIN {X 0,Y 135.338,Z 563.293,A -85,B 0,C 180,E1 -27739.386,E2 -27739.386} C_VEL
LIN {X 0,Y 137.595,Z 567.784,A -85,B 0,C 180,E1 -27742.48,E2 -27742.48} C_VEL
LIN {X 0,Y 139.614,Z 574.22,A -85,B 0,C 180,E1 -27745.157,E2 -27745.157} C_VEL
LIN {X 0,Y 140.855,Z 578.584,A -85,B 0,C 180,E1 -27746.688,E2 -27746.688} C_VEL
LIN {X 0,Y 138.84,Z 597.311,A -85,B 0,C 180,E1 -27747.434,E2 -27747.434} C_VEL
LIN {X 0,Y 135.719,Z 612.038,A -85,B 0,C 180,E1 -27748.321,E2 -27748.321} C_VEL
LIN {X 0,Y 132.798,Z 621.685,A -85,B 0,C 180,E1 -27749.166,E2 -27749.166} C_VEL
LIN {X 0,Y 128.486,Z 632.794,A -85,B 0,C 180,E1 -27750.515,E2 -27750.515} C_VEL
LIN {X 0,Y 124.206,Z 641.789,A -85,B 0,C 180,E1 -27751.925,E2 -27751.925} C_VEL
LIN {X 0,Y 119.386,Z 650.511,A -85,B 0,C 180,E1 -27753.747,E2 -27753.747} C_VEL
LIN {X 0,Y 114.681,Z 657.927,A -85,B 0,C 180,E1 -27755.709,E2 -27755.709} C_VEL
LIN {X 0,Y 108.262,Z 666.717,A -85,B 0,C 180,E1 -27758.832,E2 -27758.832} C_VEL
LIN {X 0,Y 103.388,Z 672.703,A -85,B 0,C 180,E1 -27761.606,E2 -27761.606} C_VEL
LIN {X 0,Y 97.67,Z 679.124,A -85,B 0,C 180,E1 -27765.592,E2 -27765.592} C_VEL
LIN {X 0,Y 92.722,Z 684.292,A -85,B 0,C 180,E1 -27769.89,E2 -27769.89} C_VEL
LIN {X 0,Y 87.224,Z 689.384,A -85,B 0,C 180,E1 -27775.666,E2 -27775.666} C_VEL
LIN {X 0,Y 82.775,Z 693.352,A -85,B 0,C 180,E1 -27782.162,E2 -27782.162} C_VEL
LIN {X 0,Y 79.526,Z 696.296,A -85,B 0,C 180,E1 -27789.299,E2 -27789.299} C_VEL
LIN {X 0,Y 78.056,Z 697.804,A -85,B 0,C 180,E1 -27794.329,E2 -27794.329} C_VEL
LIN {X 0,Y 76.715,Z 699.346,A -85,B 0,C 180,E1 -27804.744,E2 -27804.744} C_VEL
LIN {X 0,Y 76.786,Z 699.634,A -85,B 0,C 180,E1 -27810,E2 -27810} C_VEL
LIN {X 0,Y 77.124,Z 698.741,A -85,B 0,C 180,E1 -27820.501,E2 -27820.501} C_VEL
LIN {X 0,Y 78.057,Z 697.804,A -85,B 0,C 180,E1 -27825.671,E2 -27825.671} C_VEL
LIN {X 0,Y 81.517,Z 694.443,A -85,B 0,C 180,E1 -27835.536,E2 -27835.536} C_VEL
LIN {X 0,Y 85.647,Z 690.814,A -85,B 0,C 180,E1 -27842.233,E2 -27842.233} C_VEL
LIN {X 0,Y 90.813,Z 686.082,A -85,B 0,C 180,E1 -27848.251,E2 -27848.251} C_VEL
LIN {X 0,Y 96.755,Z 680.111,A -85,B 0,C 180,E1 -27853.631,E2 -27853.631} C_VEL
LIN {X 0,Y 102.239,Z 674.016,A -85,B 0,C 180,E1 -27857.642,E2 -27857.642} C_VEL
LIN {X 0,Y 107.036,Z 668.277,A -85,B 0,C 180,E1 -27860.488,E2 -27860.488} C_VEL
LIN {X 0,Y 112.063,Z 661.624,A -85,B 0,C 180,E1 -27863.092,E2 -27863.092} C_VEL
LIN {X 0,Y 117.342,Z 653.803,A -85,B 0,C 180,E1 -27865.439,E2 -27865.439} C_VEL
LIN {X 0,Y 122.114,Z 645.725,A -85,B 0,C 180,E1 -27867.32,E2 -27867.32} C_VEL
LIN {X 0,Y 127.048,Z 635.972,A -85,B 0,C 180,E1 -27869.028,E2 -27869.028} C_VEL
LIN {X 0,Y 130.605,Z 627.586,A -85,B 0,C 180,E1 -27870.192,E2 -27870.192} C_VEL
LIN {X 0,Y 134.258,Z 617.086,A -85,B 0,C 180,E1 -27871.259,E2 -27871.259} C_VEL
LIN {X 0,Y 136.973,Z 606.898,A -85,B 0,C 180,E1 -27872.032,E2 -27872.032} C_VEL
LIN {X 0,Y 138.959,Z 596.503,A -85,B 0,C 180,E1 -27872.583,E2 -27872.583} C_VEL
LIN {X 0,Y 140.852,Z 578.608,A -85,B 0,C 180,E1 -27873.312,E2 -27873.312} C_VEL
LIN {X 0,Y 138.335,Z 569.963,A -85,B 0,C 180,E1 -27876.519,E2 -27876.519} C_VEL
LIN {X 0,Y 137.034,Z 566.597,A -85,B 0,C 180,E1 -27878.25,E2 -27878.25} C_VEL
LIN {X 0,Y 134.388,Z 561.396,A -85,B 0,C 180,E1 -27882.102,E2 -27882.102} C_VEL
LIN {X 0,Y 132.546,Z 558.035,A -85,B 0,C 180,E1 -27885.408,E2 -27885.408} C_VEL
LIN {X 0,Y 130.787,Z 554.625,A -85,B 0,C 180,E1 -27889.644,E2 -27889.644} C_VEL
LIN {X 0,Y 129.149,Z 550.448,A -85,B 0,C 180,E1 -27898.436,E2 -27898.436} C_VEL
LIN {X 0,Y 129.117,Z 550.218,A -85,B 0,C 180,E1 -27899.995,E2 -27899.995} C_VEL
LIN {X 0,Y 129.191,Z 550.976,A -85,B 0,C 180,E1 -27903.114,E2 -27903.114} C_VEL
LIN {X 0,Y 131.092,Z 555.234,A -85,B 0,C 180,E1 -27911.605,E2 -27911.605} C_VEL
LIN {X 0,Y 133.314,Z 559.47,A -85,B 0,C 180,E1 -27916.456,E2 -27916.456} C_VEL
LIN {X 0,Y 135.509,Z 563.645,A -85,B 0,C 180,E1 -27920.032,E2 -27920.032} C_VEL
LIN {X 0,Y 137.691,Z 568.035,A -85,B 0,C 180,E1 -27922.998,E2 -27922.998} C_VEL
LIN {X 0,Y 140.777,Z 574.876,A -85,B 0,C 180,E1 -27926.6,E2 -27926.6} C_VEL
LIN {X 0,Y 141.942,Z 577.75,A -85,B 0,C 180,E1 -27927.841,E2 -27927.841} C_VEL
LIN {X 0,Y 142.897,Z 580.609,A -85,B 0,C 180,E1 -27928.849,E2 -27928.849} C_VEL
LIN {X 0,Y 143.781,Z 585.7,A -85,B 0,C 180,E1 -27930.004,E2 -27930.004} C_VEL
LIN {X 0,Y 144.052,Z 598.839,A -85,B 0,C 180,E1 -27932.09,E2 -27932.09} C_VEL
LIN {X 0,Y 144.232,Z 604.209,A -85,B 0,C 180,E1 -27933.215,E2 -27933.215} C_VEL
LIN {X 0,Y 144.414,Z 605.86,A -85,B 0,C 180,E1 -27933.673,E2 -27933.673} C_VEL
LIN {X 0,Y 146.121,Z 617.615,A -85,B 0,C 180,E1 -27937.529,E2 -27937.529} C_VEL
LIN {X 0,Y 147.721,Z 626.427,A -85,B 0,C 180,E1 -27940.851,E2 -27940.851} C_VEL
LIN {X 0,Y 150.259,Z 637.015,A -85,B 0,C 180,E1 -27945.446,E2 -27945.446} C_VEL
LIN {X 0,Y 153.122,Z 645.243,A -85,B 0,C 180,E1 -27949.501,E2 -27949.501} C_VEL
LIN {X 0,Y 156.924,Z 652.844,A -85,B 0,C 180,E1 -27953.714,E2 -27953.714} C_VEL
LIN {X 0,Y 161.322,Z 659.274,A -85,B 0,C 180,E1 -27957.627,E2 -27957.627} C_VEL
LIN {X 0,Y 168.235,Z 666.692,A -85,B 0,C 180,E1 -27962.644,E2 -27962.644} C_VEL
LIN {X 0,Y 175.723,Z 672.379,A -85,B 0,C 180,E1 -27966.898,E2 -27966.898} C_VEL
LIN {X 0,Y 185.456,Z 677.681,A -85,B 0,C 180,E1 -27971.321,E2 -27971.321} C_VEL
LIN {X 0,Y 197.154,Z 682.157,A -85,B 0,C 180,E1 -27975.55,E2 -27975.55} C_VEL
LIN {X 0,Y 207.784,Z 685.144,A -85,B 0,C 180,E1 -27978.76,E2 -27978.76} C_VEL
LIN {X 0,Y 219.948,Z 687.776,A -85,B 0,C 180,E1 -27982.087,E2 -27982.087} C_VEL
LIN {X 0,Y 226.207,Z 688.864,A -85,B 0,C 180,E1 -27983.797,E2 -27983.797} C_VEL
LIN {X 0,Y 232.563,Z 689.853,A -85,B 0,C 180,E1 -27985.705,E2 -27985.705} C_VEL
LIN {X 0,Y 234.935,Z 690.204,A -85,B 0,C 180,E1 -27986.57,E2 -27986.57} C_VEL
LIN {X 0,Y 239.034,Z 690.703,A -85,B 0,C 180,E1 -27988.372,E2 -27988.372} C_VEL
LIN {X 0,Y 241.27,Z 690.843,A -85,B 0,C 180,E1 -27990,E2 -27990} C_VEL
LIN {X 0,Y 238.865,Z 690.698,A -85,B 0,C 180,E1 -27991.686,E2 -27991.686} C_VEL
LIN {X 0,Y 234.899,Z 690.205,A -85,B 0,C 180,E1 -27993.431,E2 -27993.431} C_VEL
LIN {X 0,Y 232.562,Z 689.855,A -85,B 0,C 180,E1 -27994.291,E2 -27994.291} C_VEL
LIN {X 0,Y 226.208,Z 688.862,A -85,B 0,C 180,E1 -27996.206,E2 -27996.206} C_VEL
LIN {X 0,Y 219.956,Z 687.763,A -85,B 0,C 180,E1 -27997.927,E2 -27997.927} C_VEL
LIN {X 0,Y 205.752,Z 684.645,A -85,B 0,C 180,E1 -28001.826,E2 -28001.826} C_VEL
LIN {X 0,Y 190.724,Z 679.874,A -85,B 0,C 180,E1 -28006.663,E2 -28006.663} C_VEL
LIN {X 0,Y 180.456,Z 675.141,A -85,B 0,C 180,E1 -28010.832,E2 -28010.832} C_VEL
LIN {X 0,Y 173.065,Z 670.607,A -85,B 0,C 180,E1 -28014.489,E2 -28014.489} C_VEL
LIN {X 0,Y 165.263,Z 663.838,A -85,B 0,C 180,E1 -28019.342,E2 -28019.342} C_VEL
LIN {X 0,Y 159.164,Z 656.462,A -85,B 0,C 180,E1 -28024.123,E2 -28024.123} C_VEL
LIN {X 0,Y 154.836,Z 648.99,A -85,B 0,C 180,E1 -28028.474,E2 -28028.474} C_VEL
LIN {X 0,Y 151.85,Z 641.872,A -85,B 0,C 180,E1 -28032.231,E2 -28032.231} C_VEL
LIN {X 0,Y 148.932,Z 631.986,A -85,B 0,C 180,E1 -28036.807,E2 -28036.807} C_VEL
LIN {X 0,Y 146.991,Z 622.816,A -85,B 0,C 180,E1 -28040.549,E2 -28040.549} C_VEL
LIN {X 0,Y 145.361,Z 612.799,A -85,B 0,C 180,E1 -28044.114,E2 -28044.114} C_VEL
LIN {X 0,Y 143.902,Z 602.412,A -85,B 0,C 180,E1 -28047.318,E2 -28047.318} C_VEL
LIN {X 0,Y 142.299,Z 592.941,A -85,B 0,C 180,E1 -28050.103,E2 -28050.103} C_VEL
LIN {X 0,Y 139.886,Z 584.738,A -85,B 0,C 180,E1 -28053.022,E2 -28053.022} C_VEL
LIN {X 0,Y 136.82,Z 576.887,A -85,B 0,C 180,E1 -28056.697,E2 -28056.697} C_VEL
LIN {X 0,Y 134.209,Z 570.873,A -85,B 0,C 180,E1 -28060.395,E2 -28060.395} C_VEL
LIN {X 0,Y 132.101,Z 566.667,A -85,B 0,C 180,E1 -28063.984,E2 -28063.984} C_VEL
LIN {X 0,Y 130.94,Z 564.327,A -85,B 0,C 180,E1 -28066.423,E2 -28066.423} C_VEL
LIN {X 0,Y 129.667,Z 561.51,A -85,B 0,C 180,E1 -28069.891,E2 -28069.891} C_VEL
LIN {X 0,Y 128.258,Z 557.508,A -85,B 0,C 180,E1 -28078.435,E2 -28078.435} C_VEL
LIN {X 0,Y 128.257,Z 557.371,A -85,B 0,C 180,E1 -28080.79,E2 -28080.79} C_VEL
LIN {X 0,Y 129.894,Z 562.018,A -85,B 0,C 180,E1 -28090.428,E2 -28090.428} C_VEL
LIN {X 0,Y 131.735,Z 565.817,A -85,B 0,C 180,E1 -28094.882,E2 -28094.882} C_VEL
LIN {X 0,Y 133.83,Z 570.133,A -85,B 0,C 180,E1 -28098.631,E2 -28098.631} C_VEL
LIN {X 0,Y 135.526,Z 574.002,A -85,B 0,C 180,E1 -28101.189,E2 -28101.189} C_VEL
LIN {X 0,Y 137.409,Z 580.846,A -85,B 0,C 180,E1 -28103.983,E2 -28103.983} C_VEL
LIN {X 0,Y 137.544,Z 581.408,A -85,B 0,C 180,E1 -28104.177,E2 -28104.177} C_VEL
LIN {X 0,Y 135.389,Z 599.321,A -85,B 0,C 180,E1 -28104.873,E2 -28104.873} C_VEL
LIN {X 0,Y 132.499,Z 611.841,A -85,B 0,C 180,E1 -28105.617,E2 -28105.617} C_VEL
LIN {X 0,Y 129.49,Z 621.489,A -85,B 0,C 180,E1 -28106.425,E2 -28106.425} C_VEL
LIN {X 0,Y 125.033,Z 632.598,A -85,B 0,C 180,E1 -28107.714,E2 -28107.714} C_VEL
LIN {X 0,Y 120.602,Z 641.593,A -85,B 0,C 180,E1 -28109.061,E2 -28109.061} C_VEL
LIN {X 0,Y 115.595,Z 650.315,A -85,B 0,C 180,E1 -28110.822,E2 -28110.822} C_VEL
LIN {X 0,Y 110.683,Z 657.73,A -85,B 0,C 180,E1 -28112.72,E2 -28112.72} C_VEL
LIN {X 0,Y 103.946,Z 666.52,A -85,B 0,C 180,E1 -28115.774,E2 -28115.774} C_VEL
LIN {X 0,Y 98.807,Z 672.507,A -85,B 0,C 180,E1 -28118.519,E2 -28118.519} C_VEL
LIN {X 0,Y 92.823,Z 678.819,A -85,B 0,C 180,E1 -28122.423,E2 -28122.423} C_VEL
LIN {X 0,Y 87.384,Z 684.095,A -85,B 0,C 180,E1 -28126.873,E2 -28126.873} C_VEL
LIN {X 0,Y 81.43,Z 689.187,A -85,B 0,C 180,E1 -28132.833,E2 -28132.833} C_VEL
LIN {X 0,Y 76.549,Z 693.156,A -85,B 0,C 180,E1 -28139.672,E2 -28139.672} C_VEL
LIN {X 0,Y 72.898,Z 696.099,A -85,B 0,C 180,E1 -28147.317,E2 -28147.317} C_VEL
LIN {X 0,Y 71.22,Z 697.607,A -85,B 0,C 180,E1 -28152.78,E2 -28152.78} C_VEL
LIN {X 0,Y 69.628,Z 699.149,A -85,B 0,C 180,E1 -28164.207,E2 -28164.207} C_VEL
LIN {X 0,Y 69.683,Z 699.438,A -85,B 0,C 180,E1 -28170,E2 -28170} C_VEL
LIN {X 0,Y 70.146,Z 698.545,A -85,B 0,C 180,E1 -28181.559,E2 -28181.559} C_VEL
LIN {X 0,Y 71.221,Z 697.607,A -85,B 0,C 180,E1 -28187.219,E2 -28187.219} C_VEL
LIN {X 0,Y 75.143,Z 694.245,A -85,B 0,C 180,E1 -28197.881,E2 -28197.881} C_VEL
LIN {X 0,Y 79.71,Z 690.617,A -85,B 0,C 180,E1 -28204.967,E2 -28204.967} C_VEL
LIN {X 0,Y 85.339,Z 685.885,A -85,B 0,C 180,E1 -28211.21,E2 -28211.21} C_VEL
LIN {X 0,Y 91.699,Z 679.913,A -85,B 0,C 180,E1 -28216.723,E2 -28216.723} C_VEL
LIN {X 0,Y 97.578,Z 673.819,A -85,B 0,C 180,E1 -28220.737,E2 -28220.737} C_VEL
LIN {X 0,Y 102.643,Z 668.08,A -85,B 0,C 180,E1 -28223.563,E2 -28223.563} C_VEL
LIN {X 0,Y 107.946,Z 661.428,A -85,B 0,C 180,E1 -28226.109,E2 -28226.109} C_VEL
LIN {X 0,Y 113.462,Z 653.607,A -85,B 0,C 180,E1 -28228.395,E2 -28228.395} C_VEL
LIN {X 0,Y 118.429,Z 645.529,A -85,B 0,C 180,E1 -28230.214,E2 -28230.214} C_VEL
LIN {X 0,Y 123.547,Z 635.776,A -85,B 0,C 180,E1 -28231.849,E2 -28231.849} C_VEL
LIN {X 0,Y 127.227,Z 627.39,A -85,B 0,C 180,E1 -28232.965,E2 -28232.965} C_VEL
LIN {X 0,Y 130.994,Z 616.89,A -85,B 0,C 180,E1 -28233.981,E2 -28233.981} C_VEL
LIN {X 0,Y 133.729,Z 607.012,A -85,B 0,C 180,E1 -28234.695,E2 -28234.695} C_VEL
LIN {X 0,Y 135.834,Z 596.307,A -85,B 0,C 180,E1 -28235.244,E2 -28235.244} C_VEL
LIN {X 0,Y 137.517,Z 581.282,A -85,B 0,C 180,E1 -28235.863,E2 -28235.863} C_VEL
LIN {X 0,Y 135.527,Z 573.999,A -85,B 0,C 180,E1 -28238.811,E2 -28238.811} C_VEL
LIN {X 0,Y 133.733,Z 569.911,A -85,B 0,C 180,E1 -28241.529,E2 -28241.529} C_VEL
LIN {X 0,Y 131.825,Z 566.033,A -85,B 0,C 180,E1 -28244.931,E2 -28244.931} C_VEL
LIN {X 0,Y 130.395,Z 563.234,A -85,B 0,C 180,E1 -28248.137,E2 -28248.137} C_VEL
LIN {X 0,Y 129.549,Z 561.365,A -85,B 0,C 180,E1 -28250.629,E2 -28250.629} C_VEL
LIN {X 0,Y 128.256,Z 557.382,A -85,B 0,C 180,E1 -28259.21,E2 -28259.21} C_VEL
LIN {X 0,Y 128.269,Z 557.613,A -85,B 0,C 180,E1 -28261.958,E2 -28261.958} C_VEL
LIN {X 0,Y 129.877,Z 562.013,A -85,B 0,C 180,E1 -28270.776,E2 -28270.776} C_VEL
LIN {X 0,Y 131.821,Z 566.051,A -85,B 0,C 180,E1 -28275.455,E2 -28275.455} C_VEL
LIN {X 0,Y 133.622,Z 569.716,A -85,B 0,C 180,E1 -28278.686,E2 -28278.686} C_VEL
LIN {X 0,Y 135.81,Z 574.533,A -85,B 0,C 180,E1 -28281.956,E2 -28281.956} C_VEL
LIN {X 0,Y 138.544,Z 581.178,A -85,B 0,C 180,E1 -28285.437,E2 -28285.437} C_VEL
LIN {X 0,Y 141.095,Z 588.565,A -85,B 0,C 180,E1 -28288.439,E2 -28288.439} C_VEL
LIN {X 0,Y 143.139,Z 597.008,A -85,B 0,C 180,E1 -28291.131,E2 -28291.131} C_VEL
LIN {X 0,Y 144.414,Z 605.86,A -85,B 0,C 180,E1 -28293.673,E2 -28293.673} C_VEL
LIN {X 0,Y 144.664,Z 610.792,A -85,B 0,C 180,E1 -28294.968,E2 -28294.968} C_VEL
LIN {X 0,Y 143.819,Z 619.466,A -85,B 0,C 180,E1 -28296.849,E2 -28296.849} C_VEL
LIN {X 0,Y 142.871,Z 627.77,A -85,B 0,C 180,E1 -28298.932,E2 -28298.932} C_VEL
LIN {X 0,Y 142.876,Z 632.12,A -85,B 0,C 180,E1 -28300.499,E2 -28300.499} C_VEL
LIN {X 0,Y 145.064,Z 642.272,A -85,B 0,C 180,E1 -28305.34,E2 -28305.34} C_VEL
LIN {X 0,Y 148.647,Z 652.277,A -85,B 0,C 180,E1 -28310.923,E2 -28310.923} C_VEL
LIN {X 0,Y 152.979,Z 659.839,A -85,B 0,C 180,E1 -28315.777,E2 -28315.777} C_VEL
LIN {X 0,Y 158.89,Z 666.978,A -85,B 0,C 180,E1 -28320.886,E2 -28320.886} C_VEL
LIN {X 0,Y 165.925,Z 672.886,A -85,B 0,C 180,E1 -28325.583,E2 -28325.583} C_VEL
LIN {X 0,Y 175.284,Z 678.292,A -85,B 0,C 180,E1 -28330.417,E2 -28330.417} C_VEL
LIN {X 0,Y 185.682,Z 682.478,A -85,B 0,C 180,E1 -28334.636,E2 -28334.636} C_VEL
LIN {X 0,Y 194.311,Z 685.07,A -85,B 0,C 180,E1 -28337.551,E2 -28337.551} C_VEL
LIN {X 0,Y 206.312,Z 687.69,A -85,B 0,C 180,E1 -28341.048,E2 -28341.048} C_VEL
LIN {X 0,Y 219.066,Z 689.685,A -85,B 0,C 180,E1 -28344.477,E2 -28344.477} C_VEL
LIN {X 0,Y 225.812,Z 690.454,A -85,B 0,C 180,E1 -28346.431,E2 -28346.431} C_VEL
LIN {X 0,Y 230.637,Z 690.921,A -85,B 0,C 180,E1 -28348.254,E2 -28348.254} C_VEL
LIN {X 0,Y 231.958,Z 690.982,A -85,B 0,C 180,E1 -28348.833,E2 -28348.833} C_VEL
LIN {X 0,Y 233.784,Z 691.05,A -85,B 0,C 180,E1 -28350,E2 -28350} C_VEL
LIN {X 0,Y 231.957,Z 690.984,A -85,B 0,C 180,E1 -28351.15,E2 -28351.15} C_VEL
LIN {X 0,Y 230.603,Z 690.922,A -85,B 0,C 180,E1 -28351.746,E2 -28351.746} C_VEL
LIN {X 0,Y 225.353,Z 690.406,A -85,B 0,C 180,E1 -28353.705,E2 -28353.705} C_VEL
LIN {X 0,Y 218.89,Z 689.659,A -85,B 0,C 180,E1 -28355.575,E2 -28355.575} C_VEL
LIN {X 0,Y 206.308,Z 687.696,A -85,B 0,C 180,E1 -28358.945,E2 -28358.945} C_VEL
LIN {X 0,Y 194.017,Z 684.977,A -85,B 0,C 180,E1 -28362.553,E2 -28362.553} C_VEL
LIN {X 0,Y 180.408,Z 680.558,A -85,B 0,C 180,E1 -28367.383,E2 -28367.383} C_VEL
LIN {X 0,Y 170.843,Z 675.982,A -85,B 0,C 180,E1 -28371.73,E2 -28371.73} C_VEL
LIN {X 0,Y 163.833,Z 671.304,A -85,B 0,C 180,E1 -28375.741,E2 -28375.741} C_VEL
LIN {X 0,Y 156.188,Z 664.073,A -85,B 0,C 180,E1 -28381.255,E2 -28381.255} C_VEL
LIN {X 0,Y 151.486,Z 657.573,A -85,B 0,C 180,E1 -28385.727,E2 -28385.727} C_VEL
LIN {X 0,Y 147.656,Z 650.006,A -85,B 0,C 180,E1 -28390.406,E2 -28390.406} C_VEL
LIN {X 0,Y 144.754,Z 641.037,A -85,B 0,C 180,E1 -28395.258,E2 -28395.258} C_VEL
LIN {X 0,Y 142.896,Z 632.347,A -85,B 0,C 180,E1 -28399.412,E2 -28399.412} C_VEL
LIN {X 0,Y 141.515,Z 622.739,A -85,B 0,C 180,E1 -28403.426,E2 -28403.426} C_VEL
LIN {X 0,Y 140.634,Z 613.828,A -85,B 0,C 180,E1 -28406.659,E2 -28406.659} C_VEL
LIN {X 0,Y 139.613,Z 603.02,A -85,B 0,C 180,E1 -28410.093,E2 -28410.093} C_VEL
LIN {X 0,Y 138.427,Z 595.001,A -85,B 0,C 180,E1 -28412.714,E2 -28412.714} C_VEL
LIN {X 0,Y 136.407,Z 587.681,A -85,B 0,C 180,E1 -28415.664,E2 -28415.664} C_VEL
LIN {X 0,Y 133.765,Z 580.492,A -85,B 0,C 180,E1 -28419.435,E2 -28419.435} C_VEL
LIN {X 0,Y 131.841,Z 575.878,A -85,B 0,C 180,E1 -28422.637,E2 -28422.637} C_VEL
LIN {X 0,Y 129.889,Z 571.433,A -85,B 0,C 180,E1 -28426.711,E2 -28426.711} C_VEL
LIN {X 0,Y 128.435,Z 568.231,A -85,B 0,C 180,E1 -28430.954,E2 -28430.954} C_VEL
LIN {X 0,Y 127.377,Z 564.443,A -85,B 0,C 180,E1 -28439.215,E2 -28439.215} C_VEL
LIN {X 0,Y 127.385,Z 564.511,A -85,B 0,C 180,E1 -28440.894,E2 -28440.894} C_VEL
LIN {X 0,Y 128.719,Z 568.831,A -85,B 0,C 180,E1 -28449.63,E2 -28449.63} C_VEL
LIN {X 0,Y 130.343,Z 572.474,A -85,B 0,C 180,E1 -28453.963,E2 -28453.963} C_VEL
LIN {X 0,Y 132.364,Z 576.969,A -85,B 0,C 180,E1 -28457.881,E2 -28457.881} C_VEL
LIN {X 0,Y 133.505,Z 580.104,A -85,B 0,C 180,E1 -28459.814,E2 -28459.814} C_VEL
LIN {X 0,Y 134.449,Z 584.122,A -85,B 0,C 180,E1 -28461.468,E2 -28461.468} C_VEL
LIN {X 0,Y 132.573,Z 599.041,A -85,B 0,C 180,E1 -28462.082,E2 -28462.082} C_VEL
LIN {X 0,Y 129.589,Z 611.645,A -85,B 0,C 180,E1 -28462.787,E2 -28462.787} C_VEL
LIN {X 0,Y 126.452,Z 621.4,A -85,B 0,C 180,E1 -28463.558,E2 -28463.558} C_VEL
LIN {X 0,Y 121.899,Z 632.403,A -85,B 0,C 180,E1 -28464.763,E2 -28464.763} C_VEL
LIN {X 0,Y 117.32,Z 641.397,A -85,B 0,C 180,E1 -28466.031,E2 -28466.031} C_VEL
LIN {X 0,Y 112.121,Z 650.119,A -85,B 0,C 180,E1 -28467.702,E2 -28467.702} C_VEL
LIN {X 0,Y 107.011,Z 657.534,A -85,B 0,C 180,E1 -28469.519,E2 -28469.519} C_VEL
LIN {X 0,Y 99.948,Z 666.323,A -85,B 0,C 180,E1 -28472.457,E2 -28472.457} C_VEL
LIN {X 0,Y 94.543,Z 672.31,A -85,B 0,C 180,E1 -28475.145,E2 -28475.145} C_VEL
LIN {X 0,Y 88.168,Z 678.62,A -85,B 0,C 180,E1 -28478.997,E2 -28478.997} C_VEL
LIN {X 0,Y 81.499,Z 684.559,A -85,B 0,C 180,E1 -28484.188,E2 -28484.188} C_VEL
LIN {X 0,Y 75.872,Z 688.99,A -85,B 0,C 180,E1 -28489.579,E2 -28489.579} C_VEL
LIN {X 0,Y 70.496,Z 692.959,A -85,B 0,C 180,E1 -28496.749,E2 -28496.749} C_VEL
LIN {X 0,Y 66.359,Z 695.901,A -85,B 0,C 180,E1 -28504.936,E2 -28504.936} C_VEL
LIN {X 0,Y 64.456,Z 697.411,A -85,B 0,C 180,E1 -28510.907,E2 -28510.907} C_VEL
LIN {X 0,Y 62.561,Z 698.953,A -85,B 0,C 180,E1 -28523.55,E2 -28523.55} C_VEL
LIN {X 0,Y 62.574,Z 699.241,A -85,B 0,C 180,E1 -28530,E2 -28530} C_VEL
LIN {X 0,Y 63.182,Z 698.348,A -85,B 0,C 180,E1 -28542.854,E2 -28542.854} C_VEL
LIN {X 0,Y 64.457,Z 697.411,A -85,B 0,C 180,E1 -28549.093,E2 -28549.093} C_VEL
LIN {X 0,Y 68.926,Z 694.048,A -85,B 0,C 180,E1 -28560.652,E2 -28560.652} C_VEL
LIN {X 0,Y 73.985,Z 690.42,A -85,B 0,C 180,E1 -28568.13,E2 -28568.13} C_VEL
LIN {X 0,Y 80.107,Z 685.688,A -85,B 0,C 180,E1 -28574.576,E2 -28574.576} C_VEL
LIN {X 0,Y 85.786,Z 680.807,A -85,B 0,C 180,E1 -28579.27,E2 -28579.27} C_VEL
LIN {X 0,Y 91.937,Z 674.933,A -85,B 0,C 180,E1 -28583.384,E2 -28583.384} C_VEL
LIN {X 0,Y 97.229,Z 669.443,A -85,B 0,C 180,E1 -28586.227,E2 -28586.227} C_VEL
LIN {X 0,Y 104.149,Z 661.232,A -85,B 0,C 180,E1 -28589.357,E2 -28589.357} C_VEL
LIN {X 0,Y 109.908,Z 653.411,A -85,B 0,C 180,E1 -28591.549,E2 -28591.549} C_VEL
LIN {X 0,Y 115.067,Z 645.333,A -85,B 0,C 180,E1 -28593.284,E2 -28593.284} C_VEL
LIN {X 0,Y 120.364,Z 635.58,A -85,B 0,C 180,E1 -28594.827,E2 -28594.827} C_VEL
LIN {X 0,Y 124.147,Z 627.22,A -85,B 0,C 180,E1 -28595.886,E2 -28595.886} C_VEL
LIN {X 0,Y 127.978,Z 616.901,A -85,B 0,C 180,E1 -28596.818,E2 -28596.818} C_VEL
LIN {X 0,Y 130.824,Z 606.97,A -85,B 0,C 180,E1 -28597.492,E2 -28597.492} C_VEL
LIN {X 0,Y 133.101,Z 595.477,A -85,B 0,C 180,E1 -28598.055,E2 -28598.055} C_VEL
LIN {X 0,Y 134.449,Z 584.124,A -85,B 0,C 180,E1 -28598.532,E2 -28598.532} C_VEL
LIN {X 0,Y 133.121,Z 578.802,A -85,B 0,C 180,E1 -28600.851,E2 -28600.851} C_VEL
LIN {X 0,Y 131.003,Z 573.951,A -85,B 0,C 180,E1 -28604.635,E2 -28604.635} C_VEL
LIN {X 0,Y 129.647,Z 571.024,A -85,B 0,C 180,E1 -28607.671,E2 -28607.671} C_VEL
LIN {X 0,Y 128.437,Z 568.215,A -85,B 0,C 180,E1 -28611.341,E2 -28611.341} C_VEL
LIN {X 0,Y 127.385,Z 564.416,A -85,B 0,C 180,E1 -28619.402,E2 -28619.402} C_VEL
LIN {X 0,Y 127.383,Z 564.64,A -85,B 0,C 180,E1 -28621.576,E2 -28621.576} C_VEL
LIN {X 0,Y 128.726,Z 568.872,A -85,B 0,C 180,E1 -28630.05,E2 -28630.05} C_VEL
LIN {X 0,Y 130.35,Z 572.566,A -85,B 0,C 180,E1 -28634.385,E2 -28634.385} C_VEL
LIN {X 0,Y 132.035,Z 576.272,A -85,B 0,C 180,E1 -28637.703,E2 -28637.703} C_VEL
LIN {X 0,Y 134.371,Z 582.02,A -85,B 0,C 180,E1 -28641.471,E2 -28641.471} C_VEL
LIN {X 0,Y 136.812,Z 589.08,A -85,B 0,C 180,E1 -28644.968,E2 -28644.968} C_VEL
LIN {X 0,Y 138.753,Z 596.539,A -85,B 0,C 180,E1 -28647.83,E2 -28647.83} C_VEL
LIN {X 0,Y 139.996,Z 606.267,A -85,B 0,C 180,E1 -28650.88,E2 -28650.88} C_VEL
LIN {X 0,Y 141.04,Z 617.951,A -85,B 0,C 180,E1 -28654.785,E2 -28654.785} C_VEL
LIN {X 0,Y 142.067,Z 626.81,A -85,B 0,C 180,E1 -28658.189,E2 -28658.189} C_VEL
LIN {X 0,Y 142.876,Z 632.12,A -85,B 0,C 180,E1 -28660.499,E2 -28660.499} C_VEL
LIN {X 0,Y 143.13,Z 636.383,A -85,B 0,C 180,E1 -28662.165,E2 -28662.165} C_VEL
LIN {X 0,Y 142.105,Z 643.911,A -85,B 0,C 180,E1 -28664.782,E2 -28664.782} C_VEL
LIN {X 0,Y 141.294,Z 650.79,A -85,B 0,C 180,E1 -28667.6,E2 -28667.6} C_VEL
LIN {X 0,Y 141.846,Z 654.157,A -85,B 0,C 180,E1 -28669.507,E2 -28669.507} C_VEL
LIN {X 0,Y 145.66,Z 661.559,A -85,B 0,C 180,E1 -28674.621,E2 -28674.621} C_VEL
LIN {X 0,Y 150.655,Z 668.088,A -85,B 0,C 180,E1 -28679.645,E2 -28679.645} C_VEL
LIN {X 0,Y 156.314,Z 673.279,A -85,B 0,C 180,E1 -28684.045,E2 -28684.045} C_VEL
LIN {X 0,Y 165.193,Z 678.859,A -85,B 0,C 180,E1 -28689.373,E2 -28689.373} C_VEL
LIN {X 0,Y 175.425,Z 683.14,A -85,B 0,C 180,E1 -28694.035,E2 -28694.035} C_VEL
LIN {X 0,Y 186.716,Z 686.375,A -85,B 0,C 180,E1 -28698.117,E2 -28698.117} C_VEL
LIN {X 0,Y 199.462,Z 688.815,A -85,B 0,C 180,E1 -28701.898,E2 -28701.898} C_VEL
LIN {X 0,Y 211.584,Z 690.365,A -85,B 0,C 180,E1 -28705.15,E2 -28705.15} C_VEL
LIN {X 0,Y 218.158,Z 690.96,A -85,B 0,C 180,E1 -28706.975,E2 -28706.975} C_VEL
LIN {X 0,Y 221.888,Z 691.158,A -85,B 0,C 180,E1 -28708.185,E2 -28708.185} C_VEL
LIN {X 0,Y 224.898,Z 691.239,A -85,B 0,C 180,E1 -28709.317,E2 -28709.317} C_VEL
LIN {X 0,Y 226.136,Z 691.262,A -85,B 0,C 180,E1 -28710,E2 -28710} C_VEL
LIN {X 0,Y 224.897,Z 691.24,A -85,B 0,C 180,E1 -28710.669,E2 -28710.669} C_VEL
LIN {X 0,Y 221.877,Z 691.158,A -85,B 0,C 180,E1 -28711.815,E2 -28711.815} C_VEL
LIN {X 0,Y 218.159,Z 690.959,A -85,B 0,C 180,E1 -28713.027,E2 -28713.027} C_VEL
LIN {X 0,Y 207.973,Z 689.995,A -85,B 0,C 180,E1 -28715.819,E2 -28715.819} C_VEL
LIN {X 0,Y 192.696,Z 687.667,A -85,B 0,C 180,E1 -28720.045,E2 -28720.045} C_VEL
LIN {X 0,Y 180.952,Z 684.919,A -85,B 0,C 180,E1 -28723.855,E2 -28723.855} C_VEL
LIN {X 0,Y 170.177,Z 681.163,A -85,B 0,C 180,E1 -28728.235,E2 -28728.235} C_VEL
LIN {X 0,Y 160.588,Z 676.237,A -85,B 0,C 180,E1 -28733.224,E2 -28733.224} C_VEL
LIN {X 0,Y 153.808,Z 671.191,A -85,B 0,C 180,E1 -28737.802,E2 -28737.802} C_VEL
LIN {X 0,Y 147.367,Z 664.214,A -85,B 0,C 180,E1 -28743.437,E2 -28743.437} C_VEL
LIN {X 0,Y 143.31,Z 657.441,A -85,B 0,C 180,E1 -28748.32,E2 -28748.32} C_VEL
LIN {X 0,Y 140.265,Z 649.441,A -85,B 0,C 180,E1 -28753.414,E2 -28753.414} C_VEL
LIN {X 0,Y 138.505,Z 641.929,A -85,B 0,C 180,E1 -28757.66,E2 -28757.66} C_VEL
LIN {X 0,Y 137.296,Z 632.888,A -85,B 0,C 180,E1 -28762.108,E2 -28762.108} C_VEL
LIN {X 0,Y 136.587,Z 623.721,A -85,B 0,C 180,E1 -28766.055,E2 -28766.055} C_VEL
LIN {X 0,Y 136.129,Z 613.651,A -85,B 0,C 180,E1 -28769.783,E2 -28769.783} C_VEL
LIN {X 0,Y 135.575,Z 603.129,A -85,B 0,C 180,E1 -28773.24,E2 -28773.24} C_VEL
LIN {X 0,Y 134.602,Z 596.367,A -85,B 0,C 180,E1 -28775.829,E2 -28775.829} C_VEL
LIN {X 0,Y 132.752,Z 589.36,A -85,B 0,C 180,E1 -28779.169,E2 -28779.169} C_VEL
LIN {X 0,Y 130.644,Z 583.242,A -85,B 0,C 180,E1 -28782.997,E2 -28782.997} C_VEL
LIN {X 0,Y 128.608,Z 578.154,A -85,B 0,C 180,E1 -28787.57,E2 -28787.57} C_VEL
LIN {X 0,Y 127.295,Z 574.974,A -85,B 0,C 180,E1 -28791.872,E2 -28791.872} C_VEL
LIN {X 0,Y 126.51,Z 571.476,A -85,B 0,C 180,E1 -28799.378,E2 -28799.378} C_VEL
LIN {X 0,Y 126.508,Z 571.547,A -85,B 0,C 180,E1 -28800.539,E2 -28800.539} C_VEL
LIN {X 0,Y 127.549,Z 575.531,A -85,B 0,C 180,E1 -28808.72,E2 -28808.72} C_VEL
LIN {X 0,Y 129.018,Z 579.254,A -85,B 0,C 180,E1 -28813.117,E2 -28813.117} C_VEL
LIN {X 0,Y 130.69,Z 583.364,A -85,B 0,C 180,E1 -28816.705,E2 -28816.705} C_VEL
LIN {X 0,Y 131.463,Z 585.865,A -85,B 0,C 180,E1 -28818.209,E2 -28818.209} C_VEL
LIN {X 0,Y 131.719,Z 587.076,A -85,B 0,C 180,E1 -28818.741,E2 -28818.741} C_VEL
LIN {X 0,Y 129.504,Z 601.457,A -85,B 0,C 180,E1 -28819.315,E2 -28819.315} C_VEL
LIN {X 0,Y 126.563,Z 612.874,A -85,B 0,C 180,E1 -28819.936,E2 -28819.936} C_VEL
LIN {X 0,Y 123.605,Z 621.652,A -85,B 0,C 180,E1 -28820.585,E2 -28820.585} C_VEL
LIN {X 0,Y 119.104,Z 632.207,A -85,B 0,C 180,E1 -28821.665,E2 -28821.665} C_VEL
LIN {X 0,Y 114.382,Z 641.201,A -85,B 0,C 180,E1 -28822.834,E2 -28822.834} C_VEL
LIN {X 0,Y 108.999,Z 649.922,A -85,B 0,C 180,E1 -28824.393,E2 -28824.393} C_VEL
LIN {X 0,Y 103.687,Z 657.337,A -85,B 0,C 180,E1 -28826.092,E2 -28826.092} C_VEL
LIN {X 0,Y 96.313,Z 666.126,A -85,B 0,C 180,E1 -28828.879,E2 -28828.879} C_VEL
LIN {X 0,Y 90.624,Z 672.113,A -85,B 0,C 180,E1 -28831.455,E2 -28831.455} C_VEL
LIN {X 0,Y 83.853,Z 678.423,A -85,B 0,C 180,E1 -28835.197,E2 -28835.197} C_VEL
LIN {X 0,Y 77.514,Z 683.717,A -85,B 0,C 180,E1 -28839.629,E2 -28839.629} C_VEL
LIN {X 0,Y 70.602,Z 688.793,A -85,B 0,C 180,E1 -28845.829,E2 -28845.829} C_VEL
LIN {X 0,Y 64.665,Z 692.762,A -85,B 0,C 180,E1 -28853.291,E2 -28853.291} C_VEL
LIN {X 0,Y 59.962,Z 695.704,A -85,B 0,C 180,E1 -28862.042,E2 -28862.042} C_VEL
LIN {X 0,Y 57.766,Z 697.214,A -85,B 0,C 180,E1 -28868.593,E2 -28868.593} C_VEL
LIN {X 0,Y 55.496,Z 698.756,A -85,B 0,C 180,E1 -28882.725,E2 -28882.725} C_VEL
LIN {X 0,Y 55.486,Z 699.045,A -85,B 0,C 180,E1 -28890,E2 -28890} C_VEL
LIN {X 0,Y 56.271,Z 698.151,A -85,B 0,C 180,E1 -28904.465,E2 -28904.465} C_VEL
LIN {X 0,Y 57.767,Z 697.214,A -85,B 0,C 180,E1 -28911.406,E2 -28911.406} C_VEL
LIN {X 0,Y 62.907,Z 693.852,A -85,B 0,C 180,E1 -28923.959,E2 -28923.959} C_VEL
LIN {X 0,Y 68.512,Z 690.223,A -85,B 0,C 180,E1 -28931.818,E2 -28931.818} C_VEL
LIN {X 0,Y 75.19,Z 685.491,A -85,B 0,C 180,E1 -28938.396,E2 -28938.396} C_VEL
LIN {X 0,Y 81.29,Z 680.609,A -85,B 0,C 180,E1 -28943.102,E2 -28943.102} C_VEL
LIN {X 0,Y 87.871,Z 674.736,A -85,B 0,C 180,E1 -28947.118,E2 -28947.118} C_VEL
LIN {X 0,Y 93.45,Z 669.246,A -85,B 0,C 180,E1 -28949.867,E2 -28949.867} C_VEL
LIN {X 0,Y 100.713,Z 661.035,A -85,B 0,C 180,E1 -28952.838,E2 -28952.838} C_VEL
LIN {X 0,Y 106.71,Z 653.215,A -85,B 0,C 180,E1 -28954.9,E2 -28954.9} C_VEL
LIN {X 0,Y 112.058,Z 645.137,A -85,B 0,C 180,E1 -28956.525,E2 -28956.525} C_VEL
LIN {X 0,Y 117.522,Z 635.384,A -85,B 0,C 180,E1 -28957.959,E2 -28957.959} C_VEL
LIN {X 0,Y 121.371,Z 627.136,A -85,B 0,C 180,E1 -28958.94,E2 -28958.94} C_VEL
LIN {X 0,Y 125.074,Z 617.567,A -85,B 0,C 180,E1 -28959.752,E2 -28959.752} C_VEL
LIN {X 0,Y 128.285,Z 606.741,A -85,B 0,C 180,E1 -28960.419,E2 -28960.419} C_VEL
LIN {X 0,Y 130.527,Z 595.869,A -85,B 0,C 180,E1 -28960.923,E2 -28960.923} C_VEL
LIN {X 0,Y 131.687,Z 586.952,A -85,B 0,C 180,E1 -28961.32,E2 -28961.32} C_VEL
LIN {X 0,Y 130.934,Z 584.048,A -85,B 0,C 180,E1 -28962.825,E2 -28962.825} C_VEL
LIN {X 0,Y 129.373,Z 580.104,A -85,B 0,C 180,E1 -28966.043,E2 -28966.043} C_VEL
LIN {X 0,Y 128.067,Z 576.993,A -85,B 0,C 180,E1 -28969.468,E2 -28969.468} C_VEL
LIN {X 0,Y 127.346,Z 575.06,A -85,B 0,C 180,E1 -28972.065,E2 -28972.065} C_VEL
LIN {X 0,Y 126.52,Z 571.369,A -85,B 0,C 180,E1 -28979.995,E2 -28979.995} C_VEL
LIN {X 0,Y 126.508,Z 572.361,A -85,B 0,C 180,E1 -28982.582,E2 -28982.582} C_VEL
LIN {X 0,Y 127.547,Z 575.55,A -85,B 0,C 180,E1 -28989.11,E2 -28989.11} C_VEL
LIN {X 0,Y 129.085,Z 579.442,A -85,B 0,C 180,E1 -28993.675,E2 -28993.675} C_VEL
LIN {X 0,Y 130.695,Z 583.342,A -85,B 0,C 180,E1 -28997.097,E2 -28997.097} C_VEL
LIN {X 0,Y 132.705,Z 589.38,A -85,B 0,C 180,E1 -29000.839,E2 -29000.839} C_VEL
LIN {X 0,Y 134.559,Z 596.126,A -85,B 0,C 180,E1 -29004.077,E2 -29004.077} C_VEL
LIN {X 0,Y 135.583,Z 603.094,A -85,B 0,C 180,E1 -29006.759,E2 -29006.759} C_VEL
LIN {X 0,Y 136.125,Z 613.663,A -85,B 0,C 180,E1 -29010.217,E2 -29010.217} C_VEL
LIN {X 0,Y 136.749,Z 625.582,A -85,B 0,C 180,E1 -29014.686,E2 -29014.686} C_VEL
LIN {X 0,Y 137.715,Z 636.587,A -85,B 0,C 180,E1 -29019.632,E2 -29019.632} C_VEL
LIN {X 0,Y 139.16,Z 645.13,A -85,B 0,C 180,E1 -29024.079,E2 -29024.079} C_VEL
LIN {X 0,Y 141.846,Z 654.157,A -85,B 0,C 180,E1 -29029.507,E2 -29029.507} C_VEL
LIN {X 0,Y 142.543,Z 657.607,A -85,B 0,C 180,E1 -29031.483,E2 -29031.483} C_VEL
LIN {X 0,Y 142.456,Z 663.451,A -85,B 0,C 180,E1 -29034.723,E2 -29034.723} C_VEL
LIN {X 0,Y 142.899,Z 668.711,A -85,B 0,C 180,E1 -29038.036,E2 -29038.036} C_VEL
LIN {X 0,Y 144.388,Z 671.212,A -85,B 0,C 180,E1 -29040.04,E2 -29040.04} C_VEL
LIN {X 0,Y 153.004,Z 678.083,A -85,B 0,C 180,E1 -29046.72,E2 -29046.72} C_VEL
LIN {X 0,Y 163.378,Z 683.106,A -85,B 0,C 180,E1 -29052.475,E2 -29052.475} C_VEL
LIN {X 0,Y 173.334,Z 686.28,A -85,B 0,C 180,E1 -29056.662,E2 -29056.662} C_VEL
LIN {X 0,Y 187.616,Z 689.141,A -85,B 0,C 180,E1 -29061.383,E2 -29061.383} C_VEL
LIN {X 0,Y 197.781,Z 690.467,A -85,B 0,C 180,E1 -29064.206,E2 -29064.206} C_VEL
LIN {X 0,Y 204.837,Z 691.03,A -85,B 0,C 180,E1 -29066.065,E2 -29066.065} C_VEL
LIN {X 0,Y 212.415,Z 691.415,A -85,B 0,C 180,E1 -29068.104,E2 -29068.104} C_VEL
LIN {X 0,Y 218.049,Z 691.485,A -85,B 0,C 180,E1 -29070,E2 -29070} C_VEL
LIN {X 0,Y 210.996,Z 691.382,A -85,B 0,C 180,E1 -29072.298,E2 -29072.298} C_VEL
LIN {X 0,Y 204.318,Z 690.984,A -85,B 0,C 180,E1 -29074.086,E2 -29074.086} C_VEL
LIN {X 0,Y 191.395,Z 689.678,A -85,B 0,C 180,E1 -29077.533,E2 -29077.533} C_VEL
LIN {X 0,Y 179.03,Z 687.586,A -85,B 0,C 180,E1 -29081.319,E2 -29081.319} C_VEL
LIN {X 0,Y 167.777,Z 684.643,A -85,B 0,C 180,E1 -29085.557,E2 -29085.557} C_VEL
LIN {X 0,Y 157.569,Z 680.553,A -85,B 0,C 180,E1 -29090.516,E2 -29090.516} C_VEL
LIN {X 0,Y 150.776,Z 676.571,A -85,B 0,C 180,E1 -29094.803,E2 -29094.803} C_VEL
LIN {X 0,Y 145.08,Z 671.957,A -85,B 0,C 180,E1 -29099.323,E2 -29099.323} C_VEL
LIN {X 0,Y 139.574,Z 665.264,A -85,B 0,C 180,E1 -29105.117,E2 -29105.117} C_VEL
LIN {X 0,Y 136.077,Z 658.408,A -85,B 0,C 180,E1 -29110.386,E2 -29110.386} C_VEL
LIN {X 0,Y 133.627,Z 649.768,A -85,B 0,C 180,E1 -29116.135,E2 -29116.135} C_VEL
LIN {X 0,Y 132.434,Z 641.231,A -85,B 0,C 180,E1 -29121.078,E2 -29121.078} C_VEL
LIN {X 0,Y 132.015,Z 632.864,A -85,B 0,C 180,E1 -29125.275,E2 -29125.275} C_VEL
LIN {X 0,Y 131.983,Z 624.289,A -85,B 0,C 180,E1 -29129.022,E2 -29129.022} C_VEL
LIN {X 0,Y 132.122,Z 614.151,A -85,B 0,C 180,E1 -29132.825,E2 -29132.825} C_VEL
LIN {X 0,Y 131.982,Z 605.042,A -85,B 0,C 180,E1 -29136.05,E2 -29136.05} C_VEL
LIN {X 0,Y 131.067,Z 598.103,A -85,B 0,C 180,E1 -29139.094,E2 -29139.094} C_VEL
LIN {X 0,Y 129.6,Z 591.859,A -85,B 0,C 180,E1 -29142.652,E2 -29142.652} C_VEL
LIN {X 0,Y 128.192,Z 587.26,A -85,B 0,C 180,E1 -29146.127,E2 -29146.127} C_VEL
LIN {X 0,Y 126.795,Z 583.513,A -85,B 0,C 180,E1 -29150.232,E2 -29150.232} C_VEL
LIN {X 0,Y 126.186,Z 581.749,A -85,B 0,C 180,E1 -29152.806,E2 -29152.806} C_VEL
LIN {X 0,Y 125.645,Z 578.502,A -85,B 0,C 180,E1 -29160.005,E2 -29160.005} C_VEL
LIN {X 0,Y 126.451,Z 582.423,A -85,B 0,C 180,E1 -29167.992,E2 -29167.992} C_VEL
LIN {X 0,Y 127.673,Z 585.894,A -85,B 0,C 180,E1 -29172.119,E2 -29172.119} C_VEL
LIN {X 0,Y 129.008,Z 589.595,A -85,B 0,C 180,E1 -29175.406,E2 -29175.406} C_VEL
LIN {X 0,Y 129.196,Z 590.238,A -85,B 0,C 180,E1 -29175.853,E2 -29175.853} C_VEL
LIN {X 0,Y 127.213,Z 601.761,A -85,B 0,C 180,E1 -29176.32,E2 -29176.32} C_VEL
LIN {X 0,Y 124.31,Z 612.71,A -85,B 0,C 180,E1 -29176.858,E2 -29176.858} C_VEL
LIN {X 0,Y 121.079,Z 621.971,A -85,B 0,C 180,E1 -29177.487,E2 -29177.487} C_VEL
LIN {X 0,Y 116.67,Z 632.01,A -85,B 0,C 180,E1 -29178.425,E2 -29178.425} C_VEL
LIN {X 0,Y 111.819,Z 641.004,A -85,B 0,C 180,E1 -29179.479,E2 -29179.479} C_VEL
LIN {X 0,Y 106.26,Z 649.726,A -85,B 0,C 180,E1 -29180.898,E2 -29180.898} C_VEL
LIN {X 0,Y 100.76,Z 657.14,A -85,B 0,C 180,E1 -29182.456,E2 -29182.456} C_VEL
LIN {X 0,Y 93.086,Z 665.93,A -85,B 0,C 180,E1 -29185.043,E2 -29185.043} C_VEL
LIN {X 0,Y 87.124,Z 671.917,A -85,B 0,C 180,E1 -29187.462,E2 -29187.462} C_VEL
LIN {X 0,Y 79.953,Z 678.226,A -85,B 0,C 180,E1 -29191.015,E2 -29191.015} C_VEL
LIN {X 0,Y 72.451,Z 684.009,A -85,B 0,C 180,E1 -29195.83,E2 -29195.83} C_VEL
LIN {X 0,Y 65.686,Z 688.597,A -85,B 0,C 180,E1 -29201.5,E2 -29201.5} C_VEL
LIN {X 0,Y 59.095,Z 692.565,A -85,B 0,C 180,E1 -29209.149,E2 -29209.149} C_VEL
LIN {X 0,Y 53.757,Z 695.506,A -85,B 0,C 180,E1 -29218.47,E2 -29218.47} C_VEL
LIN {X 0,Y 51.179,Z 697.016,A -85,B 0,C 180,E1 -29225.672,E2 -29225.672} C_VEL
LIN {X 0,Y 48.443,Z 698.559,A -85,B 0,C 180,E1 -29241.658,E2 -29241.658} C_VEL
LIN {X 0,Y 48.381,Z 698.849,A -85,B 0,C 180,E1 -29250,E2 -29250} C_VEL
LIN {X 0,Y 49.396,Z 697.954,A -85,B 0,C 180,E1 -29266.532,E2 -29266.532} C_VEL
LIN {X 0,Y 51.179,Z 697.016,A -85,B 0,C 180,E1 -29274.328,E2 -29274.328} C_VEL
LIN {X 0,Y 57.145,Z 693.655,A -85,B 0,C 180,E1 -29287.946,E2 -29287.946} C_VEL
LIN {X 0,Y 63.364,Z 690.025,A -85,B 0,C 180,E1 -29296.132,E2 -29296.132} C_VEL
LIN {X 0,Y 70.655,Z 685.294,A -85,B 0,C 180,E1 -29302.726,E2 -29302.726} C_VEL
LIN {X 0,Y 77.209,Z 680.411,A -85,B 0,C 180,E1 -29307.35,E2 -29307.35} C_VEL
LIN {X 0,Y 84.22,Z 674.539,A -85,B 0,C 180,E1 -29311.187,E2 -29311.187} C_VEL
LIN {X 0,Y 90.083,Z 669.049,A -85,B 0,C 180,E1 -29313.791,E2 -29313.791} C_VEL
LIN {X 0,Y 97.663,Z 660.838,A -85,B 0,C 180,E1 -29316.564,E2 -29316.564} C_VEL
LIN {X 0,Y 103.9,Z 653.018,A -85,B 0,C 180,E1 -29318.445,E2 -29318.445} C_VEL
LIN {X 0,Y 109.427,Z 644.941,A -85,B 0,C 180,E1 -29319.931,E2 -29319.931} C_VEL
LIN {X 0,Y 115.046,Z 635.188,A -85,B 0,C 180,E1 -29321.238,E2 -29321.238} C_VEL
LIN {X 0,Y 118.947,Z 627.069,A -85,B 0,C 180,E1 -29322.125,E2 -29322.125} C_VEL
LIN {X 0,Y 122.938,Z 616.947,A -85,B 0,C 180,E1 -29322.883,E2 -29322.883} C_VEL
LIN {X 0,Y 126.246,Z 605.835,A -85,B 0,C 180,E1 -29323.5,E2 -29323.5} C_VEL
LIN {X 0,Y 128.41,Z 595.498,A -85,B 0,C 180,E1 -29323.922,E2 -29323.922} C_VEL
LIN {X 0,Y 129.15,Z 590.151,A -85,B 0,C 180,E1 -29324.207,E2 -29324.207} C_VEL
LIN {X 0,Y 127.744,Z 586.091,A -85,B 0,C 180,E1 -29327.686,E2 -29327.686} C_VEL
LIN {X 0,Y 126.37,Z 582.08,A -85,B 0,C 180,E1 -29332.405,E2 -29332.405} C_VEL
LIN {X 0,Y 125.646,Z 578.491,A -85,B 0,C 180,E1 -29339.995,E2 -29339.995} C_VEL
LIN {X 0,Y 126.449,Z 582.446,A -85,B 0,C 180,E1 -29348.384,E2 -29348.384} C_VEL
LIN {X 0,Y 127.747,Z 586.084,A -85,B 0,C 180,E1 -29352.707,E2 -29352.707} C_VEL
LIN {X 0,Y 129.032,Z 590.025,A -85,B 0,C 180,E1 -29356.102,E2 -29356.102} C_VEL
LIN {X 0,Y 130.631,Z 595.911,A -85,B 0,C 180,E1 -29359.746,E2 -29359.746} C_VEL
LIN {X 0,Y 131.649,Z 602.077,A -85,B 0,C 180,E1 -29362.765,E2 -29362.765} C_VEL
LIN {X 0,Y 132.155,Z 608.697,A -85,B 0,C 180,E1 -29365.305,E2 -29365.305} C_VEL
LIN {X 0,Y 132.032,Z 619.236,A -85,B 0,C 180,E1 -29369.012,E2 -29369.012} C_VEL
LIN {X 0,Y 131.96,Z 628.629,A -85,B 0,C 180,E1 -29372.814,E2 -29372.814} C_VEL
LIN {X 0,Y 132.212,Z 637.769,A -85,B 0,C 180,E1 -29377.123,E2 -29377.123} C_VEL
LIN {X 0,Y 133.024,Z 646.414,A -85,B 0,C 180,E1 -29381.831,E2 -29381.831} C_VEL
LIN {X 0,Y 134.728,Z 654.482,A -85,B 0,C 180,E1 -29386.904,E2 -29386.904} C_VEL
LIN {X 0,Y 137.637,Z 661.835,A -85,B 0,C 180,E1 -29392.212,E2 -29392.212} C_VEL
LIN {X 0,Y 141.76,Z 668.24,A -85,B 0,C 180,E1 -29397.428,E2 -29397.428} C_VEL
LIN {X 0,Y 144.388,Z 671.212,A -85,B 0,C 180,E1 -29400.04,E2 -29400.04} C_VEL
LIN {X 0,Y 146.055,Z 673.658,A -85,B 0,C 180,E1 -29402.066,E2 -29402.066} C_VEL
LIN {X 0,Y 147.553,Z 677.906,A -85,B 0,C 180,E1 -29405.529,E2 -29405.529} C_VEL
LIN {X 0,Y 149.63,Z 681.566,A -85,B 0,C 180,E1 -29408.972,E2 -29408.972} C_VEL
LIN {X 0,Y 152.136,Z 683.175,A -85,B 0,C 180,E1 -29410.891,E2 -29410.891} C_VEL
LIN {X 0,Y 160.138,Z 686.094,A -85,B 0,C 180,E1 -29414.892,E2 -29414.892} C_VEL
LIN {X 0,Y 171.589,Z 688.811,A -85,B 0,C 180,E1 -29419.397,E2 -29419.397} C_VEL
LIN {X 0,Y 184.533,Z 690.651,A -85,B 0,C 180,E1 -29423.439,E2 -29423.439} C_VEL
LIN {X 0,Y 197.082,Z 691.581,A -85,B 0,C 180,E1 -29426.779,E2 -29426.779} C_VEL
LIN {X 0,Y 203.865,Z 691.723,A -85,B 0,C 180,E1 -29428.538,E2 -29428.538} C_VEL
LIN {X 0,Y 208.901,Z 691.738,A -85,B 0,C 180,E1 -29430,E2 -29430} C_VEL
LIN {X 0,Y 201.83,Z 691.701,A -85,B 0,C 180,E1 -29431.996,E2 -29431.996} C_VEL
LIN {X 0,Y 190.45,Z 691.13,A -85,B 0,C 180,E1 -29434.939,E2 -29434.939} C_VEL
LIN {X 0,Y 175.79,Z 689.466,A -85,B 0,C 180,E1 -29439.202,E2 -29439.202} C_VEL
LIN {X 0,Y 165.729,Z 687.505,A -85,B 0,C 180,E1 -29442.768,E2 -29442.768} C_VEL
LIN {X 0,Y 154.854,Z 684.247,A -85,B 0,C 180,E1 -29447.637,E2 -29447.637} C_VEL
LIN {X 0,Y 146.548,Z 680.377,A -85,B 0,C 180,E1 -29452.56,E2 -29452.56} C_VEL
LIN {X 0,Y 141.148,Z 676.86,A -85,B 0,C 180,E1 -29456.623,E2 -29456.623} C_VEL
LIN {X 0,Y 135.69,Z 671.778,A -85,B 0,C 180,E1 -29461.906,E2 -29461.906} C_VEL
LIN {X 0,Y 131.368,Z 665.182,A -85,B 0,C 180,E1 -29467.908,E2 -29467.908} C_VEL
LIN {X 0,Y 128.888,Z 658.577,A -85,B 0,C 180,E1 -29473.221,E2 -29473.221} C_VEL
LIN {X 0,Y 127.477,Z 650.92,A -85,B 0,C 180,E1 -29478.587,E2 -29478.587} C_VEL
LIN {X 0,Y 127.032,Z 642.785,A -85,B 0,C 180,E1 -29483.513,E2 -29483.513} C_VEL
LIN {X 0,Y 127.221,Z 633.203,A -85,B 0,C 180,E1 -29488.477,E2 -29488.477} C_VEL
LIN {X 0,Y 127.876,Z 623.203,A -85,B 0,C 180,E1 -29492.825,E2 -29492.825} C_VEL
LIN {X 0,Y 128.526,Z 613.963,A -85,B 0,C 180,E1 -29496.3,E2 -29496.3} C_VEL
LIN {X 0,Y 128.669,Z 608.938,A -85,B 0,C 180,E1 -29498.209,E2 -29498.209} C_VEL
LIN {X 0,Y 128.166,Z 602.568,A -85,B 0,C 180,E1 -29501.212,E2 -29501.212} C_VEL
LIN {X 0,Y 127.27,Z 596.606,A -85,B 0,C 180,E1 -29504.901,E2 -29504.901} C_VEL
LIN {X 0,Y 126.176,Z 592.425,A -85,B 0,C 180,E1 -29508.56,E2 -29508.56} C_VEL
LIN {X 0,Y 125.189,Z 588.748,A -85,B 0,C 180,E1 -29513.154,E2 -29513.154} C_VEL
LIN {X 0,Y 124.76,Z 585.708,A -85,B 0,C 180,E1 -29520.005,E2 -29520.005} C_VEL
LIN {X 0,Y 125.385,Z 589.41,A -85,B 0,C 180,E1 -29527.452,E2 -29527.452} C_VEL
LIN {X 0,Y 126.291,Z 592.606,A -85,B 0,C 180,E1 -29531.236,E2 -29531.236} C_VEL
LIN {X 0,Y 126.785,Z 594.4,A -85,B 0,C 180,E1 -29532.927,E2 -29532.927} C_VEL
LIN {X 0,Y 124.295,Z 606.171,A -85,B 0,C 180,E1 -29533.4,E2 -29533.4} C_VEL
LIN {X 0,Y 120.593,Z 618.127,A -85,B 0,C 180,E1 -29533.994,E2 -29533.994} C_VEL
LIN {X 0,Y 115.45,Z 630.225,A -85,B 0,C 180,E1 -29534.899,E2 -29534.899} C_VEL
LIN {X 0,Y 109.658,Z 640.809,A -85,B 0,C 180,E1 -29535.984,E2 -29535.984} C_VEL
LIN {X 0,Y 103.933,Z 649.529,A -85,B 0,C 180,E1 -29537.229,E2 -29537.229} C_VEL
LIN {X 0,Y 98.264,Z 656.944,A -85,B 0,C 180,E1 -29538.622,E2 -29538.622} C_VEL
LIN {X 0,Y 90.306,Z 665.733,A -85,B 0,C 180,E1 -29540.952,E2 -29540.952} C_VEL
LIN {X 0,Y 84.082,Z 671.72,A -85,B 0,C 180,E1 -29543.158,E2 -29543.158} C_VEL
LIN {X 0,Y 76.525,Z 678.029,A -85,B 0,C 180,E1 -29546.438,E2 -29546.438} C_VEL
LIN {X 0,Y 67.75,Z 684.303,A -85,B 0,C 180,E1 -29551.485,E2 -29551.485} C_VEL
LIN {X 0,Y 61.205,Z 688.4,A -85,B 0,C 180,E1 -29556.508,E2 -29556.508} C_VEL
LIN {X 0,Y 53.904,Z 692.368,A -85,B 0,C 180,E1 -29564.186,E2 -29564.186} C_VEL
LIN {X 0,Y 47.817,Z 695.309,A -85,B 0,C 180,E1 -29573.991,E2 -29573.991} C_VEL
LIN {X 0,Y 44.772,Z 696.819,A -85,B 0,C 180,E1 -29581.906,E2 -29581.906} C_VEL
LIN {X 0,Y 41.424,Z 698.363,A -85,B 0,C 180,E1 -29600.232,E2 -29600.232} C_VEL
LIN {X 0,Y 41.293,Z 698.653,A -85,B 0,C 180,E1 -29610,E2 -29610} C_VEL
LIN {X 0,Y 42.614,Z 697.757,A -85,B 0,C 180,E1 -29629.259,E2 -29629.259} C_VEL
LIN {X 0,Y 44.773,Z 696.819,A -85,B 0,C 180,E1 -29638.093,E2 -29638.093} C_VEL
LIN {X 0,Y 51.721,Z 693.459,A -85,B 0,C 180,E1 -29652.797,E2 -29652.797} C_VEL
LIN {X 0,Y 58.641,Z 689.828,A -85,B 0,C 180,E1 -29661.169,E2 -29661.169} C_VEL
LIN {X 0,Y 63.875,Z 686.887,A -85,B 0,C 180,E1 -29665.608,E2 -29665.608} C_VEL
LIN {X 0,Y 72.178,Z 681.308,A -85,B 0,C 180,E1 -29671.202,E2 -29671.202} C_VEL
LIN {X 0,Y 79.511,Z 675.653,A -85,B 0,C 180,E1 -29674.957,E2 -29674.957} C_VEL
LIN {X 0,Y 87.175,Z 668.853,A -85,B 0,C 180,E1 -29677.989,E2 -29677.989} C_VEL
LIN {X 0,Y 95.056,Z 660.641,A -85,B 0,C 180,E1 -29680.504,E2 -29680.504} C_VEL
LIN {X 0,Y 101.508,Z 652.822,A -85,B 0,C 180,E1 -29682.173,E2 -29682.173} C_VEL
LIN {X 0,Y 107.2,Z 644.745,A -85,B 0,C 180,E1 -29683.495,E2 -29683.495} C_VEL
LIN {X 0,Y 112.96,Z 634.991,A -85,B 0,C 180,E1 -29684.654,E2 -29684.654} C_VEL
LIN {X 0,Y 117.559,Z 625.47,A -85,B 0,C 180,E1 -29685.534,E2 -29685.534} C_VEL
LIN {X 0,Y 121.505,Z 615.329,A -85,B 0,C 180,E1 -29686.181,E2 -29686.181} C_VEL
LIN {X 0,Y 124.505,Z 605.262,A -85,B 0,C 180,E1 -29686.656,E2 -29686.656} C_VEL
LIN {X 0,Y 126.627,Z 595.302,A -85,B 0,C 180,E1 -29687.011,E2 -29687.011} C_VEL
LIN {X 0,Y 126.717,Z 594.273,A -85,B 0,C 180,E1 -29687.178,E2 -29687.178} C_VEL
LIN {X 0,Y 125.643,Z 590.488,A -85,B 0,C 180,E1 -29691.147,E2 -29691.147} C_VEL
LIN {X 0,Y 125.138,Z 588.54,A -85,B 0,C 180,E1 -29693.95,E2 -29693.95} C_VEL
LIN {X 0,Y 124.758,Z 585.722,A -85,B 0,C 180,E1 -29700.399,E2 -29700.399} C_VEL
LIN {X 0,Y 125.264,Z 589.14,A -85,B 0,C 180,E1 -29707.45,E2 -29707.45} C_VEL
LIN {X 0,Y 126.185,Z 592.602,A -85,B 0,C 180,E1 -29711.643,E2 -29711.643} C_VEL
LIN {X 0,Y 127.319,Z 596.933,A -85,B 0,C 180,E1 -29715.298,E2 -29715.298} C_VEL
LIN {X 0,Y 128.231,Z 603.166,A -85,B 0,C 180,E1 -29719.089,E2 -29719.089} C_VEL
LIN {X 0,Y 128.671,Z 608.938,A -85,B 0,C 180,E1 -29721.794,E2 -29721.794} C_VEL
LIN {X 0,Y 128.349,Z 617.505,A -85,B 0,C 180,E1 -29724.963,E2 -29724.963} C_VEL
LIN {X 0,Y 127.538,Z 628.252,A -85,B 0,C 180,E1 -29729.273,E2 -29729.273} C_VEL
LIN {X 0,Y 127.026,Z 638.015,A -85,B 0,C 180,E1 -29733.912,E2 -29733.912} C_VEL
LIN {X 0,Y 127.085,Z 646.2,A -85,B 0,C 180,E1 -29738.466,E2 -29738.466} C_VEL
LIN {X 0,Y 127.915,Z 654.339,A -85,B 0,C 180,E1 -29743.72,E2 -29743.72} C_VEL
LIN {X 0,Y 130.015,Z 662.106,A -85,B 0,C 180,E1 -29749.56,E2 -29749.56} C_VEL
LIN {X 0,Y 133.286,Z 668.433,A -85,B 0,C 180,E1 -29755.005,E2 -29755.005} C_VEL
LIN {X 0,Y 138.114,Z 674.223,A -85,B 0,C 180,E1 -29760.612,E2 -29760.612} C_VEL
LIN {X 0,Y 145.41,Z 679.733,A -85,B 0,C 180,E1 -29766.668,E2 -29766.668} C_VEL
LIN {X 0,Y 152.136,Z 683.175,A -85,B 0,C 180,E1 -29770.891,E2 -29770.891} C_VEL
LIN {X 0,Y 154.863,Z 684.69,A -85,B 0,C 180,E1 -29772.776,E2 -29772.776} C_VEL
LIN {X 0,Y 158.3,Z 687.255,A -85,B 0,C 180,E1 -29776.057,E2 -29776.057} C_VEL
LIN {X 0,Y 162.341,Z 689.337,A -85,B 0,C 180,E1 -29779.188,E2 -29779.188} C_VEL
LIN {X 0,Y 165.901,Z 690.071,A -85,B 0,C 180,E1 -29780.794,E2 -29780.794} C_VEL
LIN {X 0,Y 176.599,Z 691.315,A -85,B 0,C 180,E1 -29784.174,E2 -29784.174} C_VEL
LIN {X 0,Y 190.567,Z 692.007,A -85,B 0,C 180,E1 -29787.887,E2 -29787.887} C_VEL
LIN {X 0,Y 198.964,Z 692.013,A -85,B 0,C 180,E1 -29790,E2 -29790} C_VEL
LIN {X 0,Y 189.895,Z 692.001,A -85,B 0,C 180,E1 -29792.292,E2 -29792.292} C_VEL
LIN {X 0,Y 172.632,Z 690.984,A -85,B 0,C 180,E1 -29797.015,E2 -29797.015} C_VEL
LIN {X 0,Y 158.143,Z 688.727,A -85,B 0,C 180,E1 -29802.146,E2 -29802.146} C_VEL
LIN {X 0,Y 147.211,Z 685.7,A -85,B 0,C 180,E1 -29807.305,E2 -29807.305} C_VEL
LIN {X 0,Y 137.825,Z 681.37,A -85,B 0,C 180,E1 -29813.398,E2 -29813.398} C_VEL
LIN {X 0,Y 131.877,Z 677.149,A -85,B 0,C 180,E1 -29818.661,E2 -29818.661} C_VEL
LIN {X 0,Y 127.346,Z 672.24,A -85,B 0,C 180,E1 -29824.134,E2 -29824.134} C_VEL
LIN {X 0,Y 123.758,Z 665.343,A -85,B 0,C 180,E1 -29830.784,E2 -29830.784} C_VEL
LIN {X 0,Y 122.156,Z 658.718,A -85,B 0,C 180,E1 -29836.346,E2 -29836.346} C_VEL
LIN {X 0,Y 121.626,Z 651.507,A -85,B 0,C 180,E1 -29841.606,E2 -29841.606} C_VEL
LIN {X 0,Y 122,Z 642.062,A -85,B 0,C 180,E1 -29847.418,E2 -29847.418} C_VEL
LIN {X 0,Y 122.909,Z 633.521,A -85,B 0,C 180,E1 -29851.882,E2 -29851.882} C_VEL
LIN {X 0,Y 124.24,Z 623.553,A -85,B 0,C 180,E1 -29856.237,E2 -29856.237} C_VEL
LIN {X 0,Y 125.349,Z 614.053,A -85,B 0,C 180,E1 -29859.933,E2 -29859.933} C_VEL
LIN {X 0,Y 125.448,Z 608.16,A -85,B 0,C 180,E1 -29862.817,E2 -29862.817} C_VEL
LIN {X 0,Y 124.953,Z 602.49,A -85,B 0,C 180,E1 -29866.383,E2 -29866.383} C_VEL
LIN {X 0,Y 124.37,Z 598.291,A -85,B 0,C 180,E1 -29870.245,E2 -29870.245} C_VEL
LIN {X 0,Y 123.824,Z 595.353,A -85,B 0,C 180,E1 -29874.305,E2 -29874.305} C_VEL
LIN {X 0,Y 123.694,Z 592.952,A -85,B 0,C 180,E1 -29880.005,E2 -29880.005} C_VEL
LIN {X 0,Y 124.01,Z 596.076,A -85,B 0,C 180,E1 -29886.513,E2 -29886.513} C_VEL
LIN {X 0,Y 124.567,Z 598.823,A -85,B 0,C 180,E1 -29889.862,E2 -29889.862} C_VEL
LIN {X 0,Y 121.445,Z 610.86,A -85,B 0,C 180,E1 -29890.334,E2 -29890.334} C_VEL
LIN {X 0,Y 117.674,Z 621.407,A -85,B 0,C 180,E1 -29890.877,E2 -29890.877} C_VEL
LIN {X 0,Y 112.991,Z 631.618,A -85,B 0,C 180,E1 -29891.583,E2 -29891.583} C_VEL
LIN {X 0,Y 107.922,Z 640.613,A -85,B 0,C 180,E1 -29892.365,E2 -29892.365} C_VEL
LIN {X 0,Y 102.05,Z 649.332,A -85,B 0,C 180,E1 -29893.407,E2 -29893.407} C_VEL
LIN {X 0,Y 96.233,Z 656.748,A -85,B 0,C 180,E1 -29894.614,E2 -29894.614} C_VEL
LIN {X 0,Y 88.016,Z 665.537,A -85,B 0,C 180,E1 -29896.629,E2 -29896.629} C_VEL
LIN {X 0,Y 81.542,Z 671.523,A -85,B 0,C 180,E1 -29898.547,E2 -29898.547} C_VEL
LIN {X 0,Y 73.629,Z 677.832,A -85,B 0,C 180,E1 -29901.465,E2 -29901.465} C_VEL
LIN {X 0,Y 65.707,Z 683.288,A -85,B 0,C 180,E1 -29905.34,E2 -29905.34} C_VEL
LIN {X 0,Y 57.261,Z 688.204,A -85,B 0,C 180,E1 -29910.78,E2 -29910.78} C_VEL
LIN {X 0,Y 49.203,Z 692.171,A -85,B 0,C 180,E1 -29918.225,E2 -29918.225} C_VEL
LIN {X 0,Y 42.252,Z 695.112,A -85,B 0,C 180,E1 -29928.292,E2 -29928.292} C_VEL
LIN {X 0,Y 38.629,Z 696.622,A -85,B 0,C 180,E1 -29936.921,E2 -29936.921} C_VEL
LIN {X 0,Y 34.427,Z 698.166,A -85,B 0,C 180,E1 -29958.221,E2 -29958.221} C_VEL
LIN {X 0,Y 34.18,Z 698.456,A -85,B 0,C 180,E1 -29970,E2 -29970} C_VEL
LIN {X 0,Y 35.974,Z 697.561,A -85,B 0,C 180,E1 -29993,E2 -29993} C_VEL
LIN {X 0,Y 38.63,Z 696.622,A -85,B 0,C 180,E1 -30003.079,E2 -30003.079} C_VEL
LIN {X 0,Y 46.734,Z 693.261,A -85,B 0,C 180,E1 -30018.756,E2 -30018.756} C_VEL
LIN {X 0,Y 54.455,Z 689.631,A -85,B 0,C 180,E1 -30027.023,E2 -30027.023} C_VEL
LIN {X 0,Y 60.131,Z 686.69,A -85,B 0,C 180,E1 -30031.233,E2 -30031.233} C_VEL
LIN {X 0,Y 69.013,Z 681.11,A -85,B 0,C 180,E1 -30036.421,E2 -30036.421} C_VEL
LIN {X 0,Y 76.77,Z 675.457,A -85,B 0,C 180,E1 -30039.775,E2 -30039.775} C_VEL
LIN {X 0,Y 84.769,Z 668.656,A -85,B 0,C 180,E1 -30042.445,E2 -30042.445} C_VEL
LIN {X 0,Y 92.925,Z 660.445,A -85,B 0,C 180,E1 -30044.641,E2 -30044.641} C_VEL
LIN {X 0,Y 99.559,Z 652.626,A -85,B 0,C 180,E1 -30046.077,E2 -30046.077} C_VEL
LIN {X 0,Y 105.403,Z 644.548,A -85,B 0,C 180,E1 -30047.199,E2 -30047.199} C_VEL
LIN {X 0,Y 111.29,Z 634.795,A -85,B 0,C 180,E1 -30048.186,E2 -30048.186} C_VEL
LIN {X 0,Y 115.853,Z 625.587,A -85,B 0,C 180,E1 -30048.915,E2 -30048.915} C_VEL
LIN {X 0,Y 119.781,Z 615.808,A -85,B 0,C 180,E1 -30049.442,E2 -30049.442} C_VEL
LIN {X 0,Y 123.07,Z 605.03,A -85,B 0,C 180,E1 -30049.872,E2 -30049.872} C_VEL
LIN {X 0,Y 124.57,Z 598.807,A -85,B 0,C 180,E1 -30050.138,E2 -30050.138} C_VEL
LIN {X 0,Y 123.892,Z 595.508,A -85,B 0,C 180,E1 -30054.298,E2 -30054.298} C_VEL
LIN {X 0,Y 123.652,Z 592.918,A -85,B 0,C 180,E1 -30060.402,E2 -30060.402} C_VEL
LIN {X 0,Y 123.927,Z 595.976,A -85,B 0,C 180,E1 -30066.712,E2 -30066.712} C_VEL
LIN {X 0,Y 124.448,Z 599.01,A -85,B 0,C 180,E1 -30070.468,E2 -30070.468} C_VEL
LIN {X 0,Y 124.999,Z 602.919,A -85,B 0,C 180,E1 -30073.923,E2 -30073.923} C_VEL
LIN {X 0,Y 125.457,Z 608.133,A -85,B 0,C 180,E1 -30077.181,E2 -30077.181} C_VEL
LIN {X 0,Y 125.35,Z 614.05,A -85,B 0,C 180,E1 -30080.067,E2 -30080.067} C_VEL
LIN {X 0,Y 124.387,Z 622.363,A -85,B 0,C 180,E1 -30083.292,E2 -30083.292} C_VEL
LIN {X 0,Y 123.326,Z 630.184,A -85,B 0,C 180,E1 -30086.579,E2 -30086.579} C_VEL
LIN {X 0,Y 122.354,Z 638.258,A -85,B 0,C 180,E1 -30090.504,E2 -30090.504} C_VEL
LIN {X 0,Y 121.693,Z 646.629,A -85,B 0,C 180,E1 -30095.27,E2 -30095.27} C_VEL
LIN {X 0,Y 121.708,Z 654.76,A -85,B 0,C 180,E1 -30100.69,E2 -30100.69} C_VEL
LIN {X 0,Y 122.815,Z 662.373,A -85,B 0,C 180,E1 -30106.632,E2 -30106.632} C_VEL
LIN {X 0,Y 124.983,Z 668.252,A -85,B 0,C 180,E1 -30111.92,E2 -30111.92} C_VEL
LIN {X 0,Y 128.763,Z 673.98,A -85,B 0,C 180,E1 -30117.766,E2 -30117.766} C_VEL
LIN {X 0,Y 133.824,Z 678.74,A -85,B 0,C 180,E1 -30123.213,E2 -30123.213} C_VEL
LIN {X 0,Y 142.332,Z 683.707,A -85,B 0,C 180,E1 -30129.779,E2 -30129.779} C_VEL
LIN {X 0,Y 148.771,Z 686.271,A -85,B 0,C 180,E1 -30133.534,E2 -30133.534} C_VEL
LIN {X 0,Y 158.139,Z 688.732,A -85,B 0,C 180,E1 -30137.861,E2 -30137.861} C_VEL
LIN {X 0,Y 165.901,Z 690.071,A -85,B 0,C 180,E1 -30140.794,E2 -30140.794} C_VEL
LIN {X 0,Y 169.632,Z 690.802,A -85,B 0,C 180,E1 -30142.343,E2 -30142.343} C_VEL
LIN {X 0,Y 174.749,Z 691.763,A -85,B 0,C 180,E1 -30145.149,E2 -30145.149} C_VEL
LIN {X 0,Y 178.993,Z 692.265,A -85,B 0,C 180,E1 -30147.322,E2 -30147.322} C_VEL
LIN {X 0,Y 182.87,Z 692.343,A -85,B 0,C 180,E1 -30148.741,E2 -30148.741} C_VEL
LIN {X 0,Y 184.354,Z 692.337,A -85,B 0,C 180,E1 -30149.147,E2 -30149.147} C_VEL
LIN {X 0,Y 187.844,Z 692.32,A -85,B 0,C 180,E1 -30150,E2 -30150} C_VEL
LIN {X 0,Y 175.927,Z 692.304,A -85,B 0,C 180,E1 -30152.997,E2 -30152.997} C_VEL
LIN {X 0,Y 160.822,Z 691.315,A -85,B 0,C 180,E1 -30157.533,E2 -30157.533} C_VEL
LIN {X 0,Y 150.569,Z 689.789,A -85,B 0,C 180,E1 -30161.445,E2 -30161.445} C_VEL
LIN {X 0,Y 138.23,Z 686.576,A -85,B 0,C 180,E1 -30167.761,E2 -30167.761} C_VEL
LIN {X 0,Y 128.309,Z 681.749,A -85,B 0,C 180,E1 -30175.159,E2 -30175.159} C_VEL
LIN {X 0,Y 122.856,Z 677.436,A -85,B 0,C 180,E1 -30180.987,E2 -30180.987} C_VEL
LIN {X 0,Y 118.556,Z 671.266,A -85,B 0,C 180,E1 -30188.141,E2 -30188.141} C_VEL
LIN {X 0,Y 116.679,Z 665.776,A -85,B 0,C 180,E1 -30193.722,E2 -30193.722} C_VEL
LIN {X 0,Y 115.855,Z 658.019,A -85,B 0,C 180,E1 -30200.445,E2 -30200.445} C_VEL
LIN {X 0,Y 116.315,Z 650.385,A -85,B 0,C 180,E1 -30206.027,E2 -30206.027} C_VEL
LIN {X 0,Y 117.329,Z 643.276,A -85,B 0,C 180,E1 -30210.516,E2 -30210.516} C_VEL
LIN {X 0,Y 119.164,Z 633.515,A -85,B 0,C 180,E1 -30215.623,E2 -30215.623} C_VEL
LIN {X 0,Y 120.994,Z 624.431,A -85,B 0,C 180,E1 -30219.609,E2 -30219.609} C_VEL
LIN {X 0,Y 122.306,Z 616.831,A -85,B 0,C 180,E1 -30222.791,E2 -30222.791} C_VEL
LIN {X 0,Y 122.553,Z 611.197,A -85,B 0,C 180,E1 -30225.899,E2 -30225.899} C_VEL
LIN {X 0,Y 122.538,Z 606.622,A -85,B 0,C 180,E1 -30229.366,E2 -30229.366} C_VEL
LIN {X 0,Y 122.222,Z 603.411,A -85,B 0,C 180,E1 -30232.987,E2 -30232.987} C_VEL
LIN {X 0,Y 122.109,Z 601.917,A -85,B 0,C 180,E1 -30235.466,E2 -30235.466} C_VEL
LIN {X 0,Y 122.264,Z 600.079,A -85,B 0,C 180,E1 -30240.005,E2 -30240.005} C_VEL
LIN {X 0,Y 122.275,Z 602.808,A -85,B 0,C 180,E1 -30245.778,E2 -30245.778} C_VEL
LIN {X 0,Y 122.34,Z 603.524,A -85,B 0,C 180,E1 -30246.772,E2 -30246.772} C_VEL
LIN {X 0,Y 119.785,Z 612.397,A -85,B 0,C 180,E1 -30247.082,E2 -30247.082} C_VEL
LIN {X 0,Y 116.226,Z 621.933,A -85,B 0,C 180,E1 -30247.479,E2 -30247.479} C_VEL
LIN {X 0,Y 111.781,Z 631.422,A -85,B 0,C 180,E1 -30248.013,E2 -30248.013} C_VEL
LIN {X 0,Y 106.627,Z 640.416,A -85,B 0,C 180,E1 -30248.635,E2 -30248.635} C_VEL
LIN {X 0,Y 100.64,Z 649.136,A -85,B 0,C 180,E1 -30249.467,E2 -30249.467} C_VEL
LIN {X 0,Y 94.692,Z 656.552,A -85,B 0,C 180,E1 -30250.456,E2 -30250.456} C_VEL
LIN {X 0,Y 86.249,Z 665.34,A -85,B 0,C 180,E1 -30252.093,E2 -30252.093} C_VEL
LIN {X 0,Y 79.561,Z 671.326,A -85,B 0,C 180,E1 -30253.669,E2 -30253.669} C_VEL
LIN {X 0,Y 71.326,Z 677.634,A -85,B 0,C 180,E1 -30256.117,E2 -30256.117} C_VEL
LIN {X 0,Y 62.196,Z 683.537,A -85,B 0,C 180,E1 -30259.826,E2 -30259.826} C_VEL
LIN {X 0,Y 53.968,Z 688.007,A -85,B 0,C 180,E1 -30264.277,E2 -30264.277} C_VEL
LIN {X 0,Y 45.142,Z 691.974,A -85,B 0,C 180,E1 -30271.1,E2 -30271.1} C_VEL
LIN {X 0,Y 37.228,Z 694.914,A -85,B 0,C 180,E1 -30280.963,E2 -30280.963} C_VEL
LIN {X 0,Y 32.893,Z 696.425,A -85,B 0,C 180,E1 -30290.135,E2 -30290.135} C_VEL
LIN {X 0,Y 27.507,Z 697.97,A -85,B 0,C 180,E1 -30315.197,E2 -30315.197} C_VEL
LIN {X 0,Y 27.07,Z 698.26,A -85,B 0,C 180,E1 -30330,E2 -30330} C_VEL
LIN {X 0,Y 29.536,Z 697.363,A -85,B 0,C 180,E1 -30358.417,E2 -30358.417} C_VEL
LIN {X 0,Y 32.893,Z 696.425,A -85,B 0,C 180,E1 -30369.865,E2 -30369.865} C_VEL
LIN {X 0,Y 42.373,Z 693.064,A -85,B 0,C 180,E1 -30386.026,E2 -30386.026} C_VEL
LIN {X 0,Y 50.93,Z 689.434,A -85,B 0,C 180,E1 -30393.76,E2 -30393.76} C_VEL
LIN {X 0,Y 60.143,Z 684.701,A -85,B 0,C 180,E1 -30399.199,E2 -30399.199} C_VEL
LIN {X 0,Y 69.707,Z 678.727,A -85,B 0,C 180,E1 -30403.295,E2 -30403.295} C_VEL
LIN {X 0,Y 77.911,Z 672.638,A -85,B 0,C 180,E1 -30405.859,E2 -30405.859} C_VEL
LIN {X 0,Y 84.57,Z 666.9,A -85,B 0,C 180,E1 -30407.54,E2 -30407.54} C_VEL
LIN {X 0,Y 91.3,Z 660.248,A -85,B 0,C 180,E1 -30408.946,E2 -30408.946} C_VEL
LIN {X 0,Y 98.088,Z 652.429,A -85,B 0,C 180,E1 -30410.123,E2 -30410.123} C_VEL
LIN {X 0,Y 104.06,Z 644.352,A -85,B 0,C 180,E1 -30411.017,E2 -30411.017} C_VEL
LIN {X 0,Y 110.057,Z 634.599,A -85,B 0,C 180,E1 -30411.803,E2 -30411.803} C_VEL
LIN {X 0,Y 114.526,Z 625.789,A -85,B 0,C 180,E1 -30412.379,E2 -30412.379} C_VEL
LIN {X 0,Y 118.685,Z 615.612,A -85,B 0,C 180,E1 -30412.815,E2 -30412.815} C_VEL
LIN {X 0,Y 121.955,Z 605.103,A -85,B 0,C 180,E1 -30413.148,E2 -30413.148} C_VEL
LIN {X 0,Y 122.33,Z 603.506,A -85,B 0,C 180,E1 -30413.283,E2 -30413.283} C_VEL
LIN {X 0,Y 122.183,Z 601.881,A -85,B 0,C 180,E1 -30415.872,E2 -30415.872} C_VEL
LIN {X 0,Y 122.265,Z 600.064,A -85,B 0,C 180,E1 -30420.407,E2 -30420.407} C_VEL
LIN {X 0,Y 122.185,Z 602.812,A -85,B 0,C 180,E1 -30426.186,E2 -30426.186} C_VEL
LIN {X 0,Y 122.484,Z 606.08,A -85,B 0,C 180,E1 -30430.116,E2 -30430.116} C_VEL
LIN {X 0,Y 122.596,Z 609.498,A -85,B 0,C 180,E1 -30432.957,E2 -30432.957} C_VEL
LIN {X 0,Y 122.481,Z 614.009,A -85,B 0,C 180,E1 -30435.811,E2 -30435.811} C_VEL
LIN {X 0,Y 121.935,Z 619.295,A -85,B 0,C 180,E1 -30438.318,E2 -30438.318} C_VEL
LIN {X 0,Y 120.051,Z 629.122,A -85,B 0,C 180,E1 -30442.358,E2 -30442.358} C_VEL
LIN {X 0,Y 118.179,Z 638.498,A -85,B 0,C 180,E1 -30446.871,E2 -30446.871} C_VEL
LIN {X 0,Y 116.754,Z 646.836,A -85,B 0,C 180,E1 -30451.65,E2 -30451.65} C_VEL
LIN {X 0,Y 115.914,Z 655.114,A -85,B 0,C 180,E1 -30457.316,E2 -30457.316} C_VEL
LIN {X 0,Y 116.145,Z 662.634,A -85,B 0,C 180,E1 -30463.438,E2 -30463.438} C_VEL
LIN {X 0,Y 117.364,Z 668.366,A -85,B 0,C 180,E1 -30468.799,E2 -30468.799} C_VEL
LIN {X 0,Y 120.214,Z 674.02,A -85,B 0,C 180,E1 -30474.922,E2 -30474.922} C_VEL
LIN {X 0,Y 124.544,Z 678.99,A -85,B 0,C 180,E1 -30480.993,E2 -30480.993} C_VEL
LIN {X 0,Y 132.216,Z 684.002,A -85,B 0,C 180,E1 -30488.156,E2 -30488.156} C_VEL
LIN {X 0,Y 139.575,Z 687.025,A -85,B 0,C 180,E1 -30493.061,E2 -30493.061} C_VEL
LIN {X 0,Y 152.509,Z 690.108,A -85,B 0,C 180,E1 -30499.378,E2 -30499.378} C_VEL
LIN {X 0,Y 162.799,Z 691.499,A -85,B 0,C 180,E1 -30503.132,E2 -30503.132} C_VEL
LIN {X 0,Y 178.802,Z 692.326,A -85,B 0,C 180,E1 -30507.747,E2 -30507.747} C_VEL
LIN {X 0,Y 184.354,Z 692.337,A -85,B 0,C 180,E1 -30509.147,E2 -30509.147} C_VEL
LIN {X 0,Y 183.285,Z 692.399,A -85,B 0,C 180,E1 -30509.27,E2 -30509.27} C_VEL
LIN {X 0,Y 182.034,Z 692.428,A -85,B 0,C 180,E1 -30509.229,E2 -30509.229} C_VEL
LIN {X 0,Y 174.881,Z 692.522,A -85,B 0,C 180,E1 -30508.404,E2 -30508.404} C_VEL
LIN {X 0,Y 165.732,Z 692.583,A -85,B 0,C 180,E1 -30506.803,E2 -30506.803} C_VEL
LIN {X 0,Y 160.779,Z 692.48,A -85,B 0,C 180,E1 -30505.693,E2 -30505.693} C_VEL
LIN {X 0,Y 156.172,Z 692.204,A -85,B 0,C 180,E1 -30504.379,E2 -30504.379} C_VEL
LIN {X 0,Y 149.086,Z 691.63,A -85,B 0,C 180,E1 -30501.836,E2 -30501.836} C_VEL
LIN {X 0,Y 137.289,Z 689.685,A -85,B 0,C 180,E1 -30496.543,E2 -30496.543} C_VEL
LIN {X 0,Y 127.022,Z 686.526,A -85,B 0,C 180,E1 -30490.135,E2 -30490.135} C_VEL
LIN {X 0,Y 118.774,Z 681.949,A -85,B 0,C 180,E1 -30482.557,E2 -30482.557} C_VEL
LIN {X 0,Y 114.375,Z 677.713,A -85,B 0,C 180,E1 -30476.426,E2 -30476.426} C_VEL
LIN {X 0,Y 111.214,Z 672.039,A -85,B 0,C 180,E1 -30469.307,E2 -30469.307} C_VEL
LIN {X 0,Y 110.063,Z 666.545,A -85,B 0,C 180,E1 -30463.339,E2 -30463.339} C_VEL
LIN {X 0,Y 110.151,Z 659.246,A -85,B 0,C 180,E1 -30456.654,E2 -30456.654} C_VEL
LIN {X 0,Y 111.523,Z 650.801,A -85,B 0,C 180,E1 -30450.268,E2 -30450.268} C_VEL
LIN {X 0,Y 113.539,Z 642.466,A -85,B 0,C 180,E1 -30445.054,E2 -30445.054} C_VEL
LIN {X 0,Y 115.835,Z 634.05,A -85,B 0,C 180,E1 -30440.682,E2 -30440.682} C_VEL
LIN {X 0,Y 118.482,Z 624.063,A -85,B 0,C 180,E1 -30436.359,E2 -30436.359} C_VEL
LIN {X 0,Y 119.57,Z 618.538,A -85,B 0,C 180,E1 -30433.593,E2 -30433.593} C_VEL
LIN {X 0,Y 119.997,Z 613.529,A -85,B 0,C 180,E1 -30430.114,E2 -30430.114} C_VEL
LIN {X 0,Y 120.127,Z 610.362,A -85,B 0,C 180,E1 -30426.714,E2 -30426.714} C_VEL
LIN {X 0,Y 120.253,Z 608.39,A -85,B 0,C 180,E1 -30423.345,E2 -30423.345} C_VEL
LIN {X 0,Y 120.469,Z 607.11,A -85,B 0,C 180,E1 -30419.995,E2 -30419.995} C_VEL
LIN {X 0,Y 120.335,Z 608.521,A -85,B 0,C 180,E1 -30416.647,E2 -30416.647} C_VEL
LIN {X 0,Y 119.344,Z 611.531,A -85,B 0,C 180,E1 -30416.367,E2 -30416.367} C_VEL
LIN {X 0,Y 115.51,Z 621.738,A -85,B 0,C 180,E1 -30416.048,E2 -30416.048} C_VEL
LIN {X 0,Y 111.006,Z 631.223,A -85,B 0,C 180,E1 -30415.672,E2 -30415.672} C_VEL
LIN {X 0,Y 105.793,Z 640.22,A -85,B 0,C 180,E1 -30415.177,E2 -30415.177} C_VEL
LIN {X 0,Y 99.721,Z 648.94,A -85,B 0,C 180,E1 -30414.547,E2 -30414.547} C_VEL
LIN {X 0,Y 93.665,Z 656.356,A -85,B 0,C 180,E1 -30413.818,E2 -30413.818} C_VEL
LIN {X 0,Y 85.045,Z 665.144,A -85,B 0,C 180,E1 -30412.591,E2 -30412.591} C_VEL
LIN {X 0,Y 78.188,Z 671.13,A -85,B 0,C 180,E1 -30411.392,E2 -30411.392} C_VEL
LIN {X 0,Y 69.686,Z 677.438,A -85,B 0,C 180,E1 -30409.512,E2 -30409.512} C_VEL
LIN {X 0,Y 60.983,Z 682.893,A -85,B 0,C 180,E1 -30406.857,E2 -30406.857} C_VEL
LIN {X 0,Y 51.453,Z 687.81,A -85,B 0,C 180,E1 -30402.965,E2 -30402.965} C_VEL
LIN {X 0,Y 41.907,Z 691.777,A -85,B 0,C 180,E1 -30397.274,E2 -30397.274} C_VEL
LIN {X 0,Y 32.992,Z 694.717,A -85,B 0,C 180,E1 -30388.438,E2 -30388.438} C_VEL
LIN {X 0,Y 27.795,Z 696.228,A -85,B 0,C 180,E1 -30379.337,E2 -30379.337} C_VEL
LIN {X 0,Y 20.754,Z 697.774,A -85,B 0,C 180,E1 -30349.794,E2 -30349.794} C_VEL
LIN {X 0,Y 19.976,Z 698.064,A -85,B 0,C 180,E1 -30330,E2 -30330} C_VEL
LIN {X 0,Y 23.511,Z 697.166,A -85,B 0,C 180,E1 -30293.285,E2 -30293.285} C_VEL
LIN {X 0,Y 27.794,Z 696.228,A -85,B 0,C 180,E1 -30280.662,E2 -30280.662} C_VEL
LIN {X 0,Y 38.843,Z 692.867,A -85,B 0,C 180,E1 -30265.223,E2 -30265.223} C_VEL
LIN {X 0,Y 48.208,Z 689.237,A -85,B 0,C 180,E1 -30258.632,E2 -30258.632} C_VEL
LIN {X 0,Y 57.988,Z 684.503,A -85,B 0,C 180,E1 -30254.17,E2 -30254.17} C_VEL
LIN {X 0,Y 66.314,Z 679.622,A -85,B 0,C 180,E1 -30251.389,E2 -30251.389} C_VEL
LIN {X 0,Y 74.775,Z 673.751,A -85,B 0,C 180,E1 -30249.296,E2 -30249.296} C_VEL
LIN {X 0,Y 81.61,Z 668.263,A -85,B 0,C 180,E1 -30247.974,E2 -30247.974} C_VEL
LIN {X 0,Y 90.204,Z 660.051,A -85,B 0,C 180,E1 -30246.6,E2 -30246.6} C_VEL
LIN {X 0,Y 97.121,Z 652.232,A -85,B 0,C 180,E1 -30245.742,E2 -30245.742} C_VEL
LIN {X 0,Y 103.191,Z 644.156,A -85,B 0,C 180,E1 -30245.092,E2 -30245.092} C_VEL
LIN {X 0,Y 109.277,Z 634.404,A -85,B 0,C 180,E1 -30244.549,E2 -30244.549} C_VEL
LIN {X 0,Y 113.603,Z 626.071,A -85,B 0,C 180,E1 -30244.168,E2 -30244.168} C_VEL
LIN {X 0,Y 118.077,Z 615.225,A -85,B 0,C 180,E1 -30243.785,E2 -30243.785} C_VEL
LIN {X 0,Y 119.715,Z 610.468,A -85,B 0,C 180,E1 -30243.633,E2 -30243.633} C_VEL
LIN {X 0,Y 120.322,Z 608.563,A -85,B 0,C 180,E1 -30243.354,E2 -30243.354} C_VEL
LIN {X 0,Y 120.471,Z 607.102,A -85,B 0,C 180,E1 -30240.005,E2 -30240.005} C_VEL
LIN {X 0,Y 120.251,Z 608.398,A -85,B 0,C 180,E1 -30236.655,E2 -30236.655} C_VEL
LIN {X 0,Y 120.136,Z 610.336,A -85,B 0,C 180,E1 -30233.286,E2 -30233.286} C_VEL
LIN {X 0,Y 119.999,Z 613.523,A -85,B 0,C 180,E1 -30229.886,E2 -30229.886} C_VEL
LIN {X 0,Y 119.718,Z 617.439,A -85,B 0,C 180,E1 -30227.101,E2 -30227.101} C_VEL
LIN {X 0,Y 118.929,Z 621.954,A -85,B 0,C 180,E1 -30224.584,E2 -30224.584} C_VEL
LIN {X 0,Y 116.977,Z 629.851,A -85,B 0,C 180,E1 -30221.212,E2 -30221.212} C_VEL
LIN {X 0,Y 114.54,Z 638.736,A -85,B 0,C 180,E1 -30216.98,E2 -30216.98} C_VEL
LIN {X 0,Y 112.453,Z 646.748,A -85,B 0,C 180,E1 -30212.407,E2 -30212.407} C_VEL
LIN {X 0,Y 110.607,Z 655.583,A -85,B 0,C 180,E1 -30206.256,E2 -30206.256} C_VEL
LIN {X 0,Y 109.908,Z 662.893,A -85,B 0,C 180,E1 -30200.114,E2 -30200.114} C_VEL
LIN {X 0,Y 110.35,Z 668.63,A -85,B 0,C 180,E1 -30194.472,E2 -30194.472} C_VEL
LIN {X 0,Y 112.154,Z 674.291,A -85,B 0,C 180,E1 -30188.03,E2 -30188.03} C_VEL
LIN {X 0,Y 116.623,Z 680.231,A -85,B 0,C 180,E1 -30180.037,E2 -30180.037} C_VEL
LIN {X 0,Y 122.631,Z 684.384,A -85,B 0,C 180,E1 -30173.528,E2 -30173.528} C_VEL
LIN {X 0,Y 127.882,Z 686.877,A -85,B 0,C 180,E1 -30169.253,E2 -30169.253} C_VEL
LIN {X 0,Y 137.293,Z 689.679,A -85,B 0,C 180,E1 -30163.464,E2 -30163.464} C_VEL
LIN {X 0,Y 149.201,Z 691.642,A -85,B 0,C 180,E1 -30158.124,E2 -30158.124} C_VEL
LIN {X 0,Y 166.865,Z 692.649,A -85,B 0,C 180,E1 -30152.414,E2 -30152.414} C_VEL
LIN {X 0,Y 176.225,Z 692.641,A -85,B 0,C 180,E1 -30150,E2 -30150} C_VEL
LIN {X 0,Y 157.75,Z 692.317,A -85,B 0,C 180,E1 -30144.888,E2 -30144.888} C_VEL
LIN {X 0,Y 156.172,Z 692.204,A -85,B 0,C 180,E1 -30144.379,E2 -30144.379} C_VEL
LIN {X 0,Y 151.395,Z 691.971,A -85,B 0,C 180,E1 -30143.081,E2 -30143.081} C_VEL
LIN {X 0,Y 135.752,Z 691.375,A -85,B 0,C 180,E1 -30139.654,E2 -30139.654} C_VEL
LIN {X 0,Y 131.249,Z 690.893,A -85,B 0,C 180,E1 -30138.042,E2 -30138.042} C_VEL
LIN {X 0,Y 129.979,Z 690.679,A -85,B 0,C 180,E1 -30137.394,E2 -30137.394} C_VEL
LIN {X 0,Y 119.38,Z 687.77,A -85,B 0,C 180,E1 -30130.361,E2 -30130.361} C_VEL
LIN {X 0,Y 111.274,Z 683.514,A -85,B 0,C 180,E1 -30122.143,E2 -30122.143} C_VEL
LIN {X 0,Y 105.892,Z 677.522,A -85,B 0,C 180,E1 -30112.78,E2 -30112.78} C_VEL
LIN {X 0,Y 103.973,Z 671.759,A -85,B 0,C 180,E1 -30105.185,E2 -30105.185} C_VEL
LIN {X 0,Y 103.867,Z 666.196,A -85,B 0,C 180,E1 -30098.962,E2 -30098.962} C_VEL
LIN {X 0,Y 105.005,Z 659.171,A -85,B 0,C 180,E1 -30092.366,E2 -30092.366} C_VEL
LIN {X 0,Y 107.436,Z 650.711,A -85,B 0,C 180,E1 -30085.96,E2 -30085.96} C_VEL
LIN {X 0,Y 109.83,Z 643.76,A -85,B 0,C 180,E1 -30081.581,E2 -30081.581} C_VEL
LIN {X 0,Y 113.097,Z 634.38,A -85,B 0,C 180,E1 -30076.719,E2 -30076.719} C_VEL
LIN {X 0,Y 115.908,Z 625.867,A -85,B 0,C 180,E1 -30072.925,E2 -30072.925} C_VEL
LIN {X 0,Y 116.838,Z 621.638,A -85,B 0,C 180,E1 -30070.391,E2 -30070.391} C_VEL
LIN {X 0,Y 117.443,Z 618.499,A -85,B 0,C 180,E1 -30067.751,E2 -30067.751} C_VEL
LIN {X 0,Y 117.759,Z 615.991,A -85,B 0,C 180,E1 -30064.552,E2 -30064.552} C_VEL
